LIN {X 0,Y 311.633,Z 530.648,A -85,B 0,C 180,E1 -15771.834,E2 -15771.834} C_VEL
LIN {X 0,Y 312.402,Z 526.953,A -85,B 0,C 180,E1 -15773.886,E2 -15773.886} C_VEL
LIN {X 0,Y 313.36,Z 522.43,A -85,B 0,C 180,E1 -15775.791,E2 -15775.791} C_VEL
LIN {X 0,Y 314.734,Z 515.773,A -85,B 0,C 180,E1 -15777.963,E2 -15777.963} C_VEL
LIN {X 0,Y 316.431,Z 507.874,A -85,B 0,C 180,E1 -15779.981,E2 -15779.981} C_VEL
LIN {X 0,Y 317.947,Z 499.641,A -85,B 0,C 180,E1 -15781.665,E2 -15781.665} C_VEL
LIN {X 0,Y 319.87,Z 489.513,A -85,B 0,C 180,E1 -15783.316,E2 -15783.316} C_VEL
LIN {X 0,Y 321.561,Z 479.498,A -85,B 0,C 180,E1 -15784.627,E2 -15784.627} C_VEL
LIN {X 0,Y 323.116,Z 468.579,A -85,B 0,C 180,E1 -15785.769,E2 -15785.769} C_VEL
LIN {X 0,Y 324.604,Z 456.019,A -85,B 0,C 180,E1 -15786.766,E2 -15786.766} C_VEL
LIN {X 0,Y 325.709,Z 443.241,A -85,B 0,C 180,E1 -15787.508,E2 -15787.508} C_VEL
LIN {X 0,Y 326.456,Z 430.389,A -85,B 0,C 180,E1 -15787.992,E2 -15787.992} C_VEL
LIN {X 0,Y 328.636,Z 357.959,A -85,B 0,C 180,E1 -15789.604,E2 -15789.604} C_VEL
LIN {X 0,Y 327.104,Z 351.684,A -85,B 0,C 180,E1 -15789.919,E2 -15789.919} C_VEL
LIN {X 0,Y 320.533,Z 336.835,A -85,B 0,C 180,E1 -15791,E2 -15791} C_VEL
LIN {X 0,Y 316.025,Z 327.77,A -85,B 0,C 180,E1 -15791.748,E2 -15791.748} C_VEL
LIN {X 0,Y 314.284,Z 325.682,A -85,B 0,C 180,E1 -15792.062,E2 -15792.062} C_VEL
LIN {X 0,Y 311.54,Z 323.906,A -85,B 0,C 180,E1 -15792.658,E2 -15792.658} C_VEL
LIN {X 0,Y 307.401,Z 321.61,A -85,B 0,C 180,E1 -15793.918,E2 -15793.918} C_VEL
LIN {X 0,Y 305.899,Z 319.461,A -85,B 0,C 180,E1 -15794.842,E2 -15794.842} C_VEL
LIN {X 0,Y 305.396,Z 317.446,A -85,B 0,C 180,E1 -15795.615,E2 -15795.615} C_VEL
LIN {X 0,Y 305.402,Z 317.444,A -85,B 0,C 180,E1 -15799.41,E2 -15799.41} C_VEL
LIN {X 0,Y 305.462,Z 317.438,A -85,B 0,C 180,E1 -15803.259,E2 -15803.259} C_VEL
LIN {X 0,Y 305.457,Z 317.413,A -85,B 0,C 180,E1 -15806.483,E2 -15806.483} C_VEL
LIN {X 0,Y 305.422,Z 317.44,A -85,B 0,C 180,E1 -15809.587,E2 -15809.587} C_VEL
LIN {X 0,Y 305.443,Z 317.437,A -85,B 0,C 180,E1 -15812.601,E2 -15812.601} C_VEL
LIN {X 0,Y 305.45,Z 317.436,A -85,B 0,C 180,E1 -15815.534,E2 -15815.534} C_VEL
LIN {X 0,Y 305.47,Z 317.436,A -85,B 0,C 180,E1 -15819.812,E2 -15819.812} C_VEL
LIN {X 0,Y 305.505,Z 317.43,A -85,B 0,C 180,E1 -15823.975,E2 -15823.975} C_VEL
LIN {X 0,Y 305.56,Z 317.41,A -85,B 0,C 180,E1 -15826.703,E2 -15826.703} C_VEL
LIN {X 0,Y 305.744,Z 317.386,A -85,B 0,C 180,E1 -15831.262,E2 -15831.262} C_VEL
LIN {X 0,Y 305.773,Z 317.392,A -85,B 0,C 180,E1 -15833.401,E2 -15833.401} C_VEL
LIN {X 0,Y 305.922,Z 317.377,A -85,B 0,C 180,E1 -15838.684,E2 -15838.684} C_VEL
LIN {X 0,Y 305.936,Z 317.367,A -85,B 0,C 180,E1 -15841.317,E2 -15841.317} C_VEL
LIN {X 0,Y 305.784,Z 317.385,A -85,B 0,C 180,E1 -15846.599,E2 -15846.599} C_VEL
LIN {X 0,Y 305.686,Z 317.401,A -85,B 0,C 180,E1 -15849.262,E2 -15849.262} C_VEL
LIN {X 0,Y 305.578,Z 317.405,A -85,B 0,C 180,E1 -15853.297,E2 -15853.297} C_VEL
LIN {X 0,Y 305.544,Z 317.42,A -85,B 0,C 180,E1 -15856.023,E2 -15856.023} C_VEL
LIN {X 0,Y 305.539,Z 317.417,A -85,B 0,C 180,E1 -15859.429,E2 -15859.429} C_VEL
LIN {X 0,Y 305.464,Z 317.423,A -85,B 0,C 180,E1 -15863.033,E2 -15863.033} C_VEL
LIN {X 0,Y 305.446,Z 317.433,A -85,B 0,C 180,E1 -15866.192,E2 -15866.192} C_VEL
LIN {X 0,Y 305.442,Z 317.435,A -85,B 0,C 180,E1 -15869.035,E2 -15869.035} C_VEL
LIN {X 0,Y 305.43,Z 317.432,A -85,B 0,C 180,E1 -15871.954,E2 -15871.954} C_VEL
LIN {X 0,Y 305.456,Z 317.431,A -85,B 0,C 180,E1 -15875.114,E2 -15875.114} C_VEL
LIN {X 0,Y 305.405,Z 317.437,A -85,B 0,C 180,E1 -15878.521,E2 -15878.521} C_VEL
LIN {X 0,Y 305.431,Z 317.422,A -85,B 0,C 180,E1 -15882.583,E2 -15882.583} C_VEL
LIN {X 0,Y 305.421,Z 317.445,A -85,B 0,C 180,E1 -15886.346,E2 -15886.346} C_VEL
LIN {X 0,Y 305.454,Z 317.439,A -85,B 0,C 180,E1 -15889.894,E2 -15889.894} C_VEL
LIN {X 0,Y 305.506,Z 317.511,A -85,B 0,C 180,E1 -15894.085,E2 -15894.085} C_VEL
LIN {X 0,Y 307.997,Z 327.276,A -85,B 0,C 180,E1 -15897.595,E2 -15897.595} C_VEL
LIN {X 0,Y 310.234,Z 336.989,A -85,B 0,C 180,E1 -15900.854,E2 -15900.854} C_VEL
LIN {X 0,Y 310.749,Z 339.325,A -85,B 0,C 180,E1 -15901.605,E2 -15901.605} C_VEL
LIN {X 0,Y 315.733,Z 351.12,A -85,B 0,C 180,E1 -15902.503,E2 -15902.503} C_VEL
LIN {X 0,Y 320.684,Z 375.641,A -85,B 0,C 180,E1 -15903.684,E2 -15903.684} C_VEL
LIN {X 0,Y 321.841,Z 383.222,A -85,B 0,C 180,E1 -15904,E2 -15904} C_VEL
LIN {X 0,Y 319.871,Z 448.323,A -85,B 0,C 180,E1 -15905.5,E2 -15905.5} C_VEL
LIN {X 0,Y 318.913,Z 461.298,A -85,B 0,C 180,E1 -15906.028,E2 -15906.028} C_VEL
LIN {X 0,Y 317.608,Z 472.761,A -85,B 0,C 180,E1 -15906.702,E2 -15906.702} C_VEL
LIN {X 0,Y 316.083,Z 484.24,A -85,B 0,C 180,E1 -15907.62,E2 -15907.62} C_VEL
LIN {X 0,Y 314.465,Z 494.745,A -85,B 0,C 180,E1 -15908.706,E2 -15908.706} C_VEL
LIN {X 0,Y 312.395,Z 505.538,A -85,B 0,C 180,E1 -15910.108,E2 -15910.108} C_VEL
LIN {X 0,Y 310.427,Z 515.474,A -85,B 0,C 180,E1 -15911.738,E2 -15911.738} C_VEL
LIN {X 0,Y 308.824,Z 523.96,A -85,B 0,C 180,E1 -15913.474,E2 -15913.474} C_VEL
LIN {X 0,Y 307.146,Z 531.649,A -85,B 0,C 180,E1 -15915.423,E2 -15915.423} C_VEL
LIN {X 0,Y 305.816,Z 537.841,A -85,B 0,C 180,E1 -15917.391,E2 -15917.391} C_VEL
LIN {X 0,Y 304.865,Z 542.782,A -85,B 0,C 180,E1 -15919.374,E2 -15919.374} C_VEL
LIN {X 0,Y 304.196,Z 546.618,A -85,B 0,C 180,E1 -15921.364,E2 -15921.364} C_VEL
LIN {X 0,Y 303.827,Z 549.45,A -85,B 0,C 180,E1 -15923.36,E2 -15923.36} C_VEL
LIN {X 0,Y 303.597,Z 551.759,A -85,B 0,C 180,E1 -15926.019,E2 -15926.019} C_VEL
LIN {X 0,Y 303.602,Z 552.335,A -85,B 0,C 180,E1 -15927.348,E2 -15927.348} C_VEL
LIN {X 0,Y 303.565,Z 552.482,A -85,B 0,C 180,E1 -15928.675,E2 -15928.675} C_VEL
LIN {X 0,Y 303.605,Z 552.23,A -85,B 0,C 180,E1 -15930.001,E2 -15930.001} C_VEL
LIN {X 0,Y 303.58,Z 551.589,A -85,B 0,C 180,E1 -15931.328,E2 -15931.328} C_VEL
LIN {X 0,Y 303.616,Z 550.557,A -85,B 0,C 180,E1 -15932.655,E2 -15932.655} C_VEL
LIN {X 0,Y 303.642,Z 549.076,A -85,B 0,C 180,E1 -15933.983,E2 -15933.983} C_VEL
LIN {X 0,Y 303.675,Z 546.624,A -85,B 0,C 180,E1 -15935.638,E2 -15935.638} C_VEL
LIN {X 0,Y 303.945,Z 541.933,A -85,B 0,C 180,E1 -15937.976,E2 -15937.976} C_VEL
LIN {X 0,Y 304.473,Z 535.613,A -85,B 0,C 180,E1 -15940.306,E2 -15940.306} C_VEL
LIN {X 0,Y 305.198,Z 528.715,A -85,B 0,C 180,E1 -15942.3,E2 -15942.3} C_VEL
LIN {X 0,Y 306.095,Z 521.67,A -85,B 0,C 180,E1 -15943.952,E2 -15943.952} C_VEL
LIN {X 0,Y 307.18,Z 513.169,A -85,B 0,C 180,E1 -15945.596,E2 -15945.596} C_VEL
LIN {X 0,Y 308.266,Z 502.616,A -85,B 0,C 180,E1 -15947.241,E2 -15947.241} C_VEL
LIN {X 0,Y 309.485,Z 492.181,A -85,B 0,C 180,E1 -15948.538,E2 -15948.538} C_VEL
LIN {X 0,Y 310.709,Z 480.737,A -85,B 0,C 180,E1 -15949.662,E2 -15949.662} C_VEL
LIN {X 0,Y 311.763,Z 468.97,A -85,B 0,C 180,E1 -15950.539,E2 -15950.539} C_VEL
LIN {X 0,Y 312.642,Z 455.38,A -85,B 0,C 180,E1 -15951.254,E2 -15951.254} C_VEL
LIN {X 0,Y 313.173,Z 441.759,A -85,B 0,C 180,E1 -15951.691,E2 -15951.691} C_VEL
LIN {X 0,Y 314.389,Z 380.153,A -85,B 0,C 180,E1 -15953.088,E2 -15953.088} C_VEL
LIN {X 0,Y 308.852,Z 339.998,A -85,B 0,C 180,E1 -15954.446,E2 -15954.446} C_VEL
LIN {X 0,Y 309.01,Z 335.76,A -85,B 0,C 180,E1 -15955.604,E2 -15955.604} C_VEL
LIN {X 0,Y 307.372,Z 326.429,A -85,B 0,C 180,E1 -15958.324,E2 -15958.324} C_VEL
LIN {X 0,Y 305.509,Z 317.433,A -85,B 0,C 180,E1 -15961.076,E2 -15961.076} C_VEL
LIN {X 0,Y 305.466,Z 317.433,A -85,B 0,C 180,E1 -15965.114,E2 -15965.114} C_VEL
LIN {X 0,Y 305.416,Z 317.441,A -85,B 0,C 180,E1 -15968.52,E2 -15968.52} C_VEL
LIN {X 0,Y 305.44,Z 317.439,A -85,B 0,C 180,E1 -15972.582,E2 -15972.582} C_VEL
LIN {X 0,Y 305.43,Z 317.442,A -85,B 0,C 180,E1 -15976.345,E2 -15976.345} C_VEL
LIN {X 0,Y 305.463,Z 317.433,A -85,B 0,C 180,E1 -15979.893,E2 -15979.893} C_VEL
LIN {X 0,Y 305.485,Z 317.429,A -85,B 0,C 180,E1 -15983.632,E2 -15983.632} C_VEL
LIN {X 0,Y 305.47,Z 317.433,A -85,B 0,C 180,E1 -15986.483,E2 -15986.483} C_VEL
LIN {X 0,Y 305.439,Z 317.435,A -85,B 0,C 180,E1 -15989.588,E2 -15989.588} C_VEL
LIN {X 0,Y 305.476,Z 317.432,A -85,B 0,C 180,E1 -15992.604,E2 -15992.604} C_VEL
LIN {X 0,Y 305.493,Z 317.43,A -85,B 0,C 180,E1 -15995.537,E2 -15995.537} C_VEL
LIN {X 0,Y 305.489,Z 317.425,A -85,B 0,C 180,E1 -15999.813,E2 -15999.813} C_VEL
LIN {X 0,Y 305.555,Z 317.422,A -85,B 0,C 180,E1 -16003.978,E2 -16003.978} C_VEL
LIN {X 0,Y 305.591,Z 317.415,A -85,B 0,C 180,E1 -16006.704,E2 -16006.704} C_VEL
LIN {X 0,Y 305.76,Z 317.389,A -85,B 0,C 180,E1 -16011.258,E2 -16011.258} C_VEL
LIN {X 0,Y 305.811,Z 317.387,A -85,B 0,C 180,E1 -16013.401,E2 -16013.401} C_VEL
LIN {X 0,Y 305.953,Z 317.37,A -85,B 0,C 180,E1 -16018.683,E2 -16018.683} C_VEL
LIN {X 0,Y 305.954,Z 317.365,A -85,B 0,C 180,E1 -16021.316,E2 -16021.316} C_VEL
LIN {X 0,Y 305.67,Z 317.403,A -85,B 0,C 180,E1 -16025.277,E2 -16025.277} C_VEL
LIN {X 0,Y 305.75,Z 317.397,A -85,B 0,C 180,E1 -16027.927,E2 -16027.927} C_VEL
LIN {X 0,Y 305.603,Z 317.413,A -85,B 0,C 180,E1 -16031.945,E2 -16031.945} C_VEL
LIN {X 0,Y 305.612,Z 317.408,A -85,B 0,C 180,E1 -16035.014,E2 -16035.014} C_VEL
LIN {X 0,Y 305.521,Z 317.427,A -85,B 0,C 180,E1 -16038.786,E2 -16038.786} C_VEL
LIN {X 0,Y 305.49,Z 317.432,A -85,B 0,C 180,E1 -16043.039,E2 -16043.039} C_VEL
LIN {X 0,Y 305.481,Z 317.425,A -85,B 0,C 180,E1 -16046.2,E2 -16046.2} C_VEL
LIN {X 0,Y 305.466,Z 317.428,A -85,B 0,C 180,E1 -16049.038,E2 -16049.038} C_VEL
LIN {X 0,Y 305.44,Z 317.434,A -85,B 0,C 180,E1 -16051.952,E2 -16051.952} C_VEL
LIN {X 0,Y 305.465,Z 317.433,A -85,B 0,C 180,E1 -16055.112,E2 -16055.112} C_VEL
LIN {X 0,Y 305.443,Z 317.427,A -85,B 0,C 180,E1 -16058.526,E2 -16058.526} C_VEL
LIN {X 0,Y 305.457,Z 317.432,A -85,B 0,C 180,E1 -16062.585,E2 -16062.585} C_VEL
LIN {X 0,Y 305.427,Z 317.434,A -85,B 0,C 180,E1 -16066.344,E2 -16066.344} C_VEL
LIN {X 0,Y 305.459,Z 317.435,A -85,B 0,C 180,E1 -16069.891,E2 -16069.891} C_VEL
LIN {X 0,Y 305.465,Z 317.432,A -85,B 0,C 180,E1 -16073.635,E2 -16073.635} C_VEL
LIN {X 0,Y 305.467,Z 317.435,A -85,B 0,C 180,E1 -16076.482,E2 -16076.482} C_VEL
LIN {X 0,Y 305.444,Z 317.434,A -85,B 0,C 180,E1 -16079.588,E2 -16079.588} C_VEL
LIN {X 0,Y 305.473,Z 317.436,A -85,B 0,C 180,E1 -16082.603,E2 -16082.603} C_VEL
LIN {X 0,Y 305.493,Z 317.428,A -85,B 0,C 180,E1 -16085.536,E2 -16085.536} C_VEL
LIN {X 0,Y 305.514,Z 317.427,A -85,B 0,C 180,E1 -16089.814,E2 -16089.814} C_VEL
LIN {X 0,Y 305.545,Z 317.426,A -85,B 0,C 180,E1 -16092.6,E2 -16092.6} C_VEL
LIN {X 0,Y 305.627,Z 317.415,A -85,B 0,C 180,E1 -16095.347,E2 -16095.347} C_VEL
LIN {X 0,Y 305.649,Z 317.603,A -85,B 0,C 180,E1 -16097.381,E2 -16097.381} C_VEL
LIN {X 0,Y 307.014,Z 324.322,A -85,B 0,C 180,E1 -16099.514,E2 -16099.514} C_VEL
LIN {X 0,Y 311.663,Z 338.303,A -85,B 0,C 180,E1 -16100.189,E2 -16100.189} C_VEL
LIN {X 0,Y 314.867,Z 355.721,A -85,B 0,C 180,E1 -16100.816,E2 -16100.816} C_VEL
LIN {X 0,Y 313.102,Z 432.447,A -85,B 0,C 180,E1 -16102.583,E2 -16102.583} C_VEL
LIN {X 0,Y 312.504,Z 444.643,A -85,B 0,C 180,E1 -16103.097,E2 -16103.097} C_VEL
LIN {X 0,Y 311.661,Z 457.936,A -85,B 0,C 180,E1 -16103.931,E2 -16103.931} C_VEL
LIN {X 0,Y 310.641,Z 469.932,A -85,B 0,C 180,E1 -16104.971,E2 -16104.971} C_VEL
LIN {X 0,Y 309.465,Z 481.372,A -85,B 0,C 180,E1 -16106.255,E2 -16106.255} C_VEL
LIN {X 0,Y 308.21,Z 491.721,A -85,B 0,C 180,E1 -16107.712,E2 -16107.712} C_VEL
LIN {X 0,Y 307.015,Z 501.006,A -85,B 0,C 180,E1 -16109.343,E2 -16109.343} C_VEL
LIN {X 0,Y 305.866,Z 510.01,A -85,B 0,C 180,E1 -16111.315,E2 -16111.315} C_VEL
LIN {X 0,Y 305.023,Z 517.26,A -85,B 0,C 180,E1 -16113.301,E2 -16113.301} C_VEL
LIN {X 0,Y 304.453,Z 523.042,A -85,B 0,C 180,E1 -16115.297,E2 -16115.297} C_VEL
LIN {X 0,Y 304.041,Z 527.598,A -85,B 0,C 180,E1 -16117.303,E2 -16117.303} C_VEL
LIN {X 0,Y 303.699,Z 531.071,A -85,B 0,C 180,E1 -16119.321,E2 -16119.321} C_VEL
LIN {X 0,Y 303.515,Z 532.798,A -85,B 0,C 180,E1 -16120.674,E2 -16120.674} C_VEL
LIN {X 0,Y 303.468,Z 534.112,A -85,B 0,C 180,E1 -16122.029,E2 -16122.029} C_VEL
LIN {X 0,Y 303.461,Z 535.04,A -85,B 0,C 180,E1 -16123.421,E2 -16123.421} C_VEL
LIN {X 0,Y 303.436,Z 535.485,A -85,B 0,C 180,E1 -16124.759,E2 -16124.759} C_VEL
LIN {X 0,Y 303.462,Z 535.535,A -85,B 0,C 180,E1 -16126.134,E2 -16126.134} C_VEL
LIN {X 0,Y 303.807,Z 534.666,A -85,B 0,C 180,E1 -16128.477,E2 -16128.477} C_VEL
LIN {X 0,Y 304.097,Z 533.152,A -85,B 0,C 180,E1 -16130.282,E2 -16130.282} C_VEL
LIN {X 0,Y 304.9,Z 529.796,A -85,B 0,C 180,E1 -16132.78,E2 -16132.78} C_VEL
LIN {X 0,Y 305.907,Z 525.122,A -85,B 0,C 180,E1 -16135.151,E2 -16135.151} C_VEL
LIN {X 0,Y 307.165,Z 519.622,A -85,B 0,C 180,E1 -16137.231,E2 -16137.231} C_VEL
LIN {X 0,Y 308.709,Z 512.642,A -85,B 0,C 180,E1 -16139.304,E2 -16139.304} C_VEL
LIN {X 0,Y 310.269,Z 505.274,A -85,B 0,C 180,E1 -16141.06,E2 -16141.06} C_VEL
LIN {X 0,Y 312.033,Z 496.703,A -85,B 0,C 180,E1 -16142.72,E2 -16142.72} C_VEL
LIN {X 0,Y 313.87,Z 486.979,A -85,B 0,C 180,E1 -16144.233,E2 -16144.233} C_VEL
LIN {X 0,Y 315.659,Z 476.269,A -85,B 0,C 180,E1 -16145.566,E2 -16145.566} C_VEL
LIN {X 0,Y 317.333,Z 464.433,A -85,B 0,C 180,E1 -16146.723,E2 -16146.723} C_VEL
LIN {X 0,Y 318.661,Z 453.162,A -85,B 0,C 180,E1 -16147.555,E2 -16147.555} C_VEL
LIN {X 0,Y 319.643,Z 440.318,A -85,B 0,C 180,E1 -16148.247,E2 -16148.247} C_VEL
LIN {X 0,Y 320.384,Z 426.831,A -85,B 0,C 180,E1 -16148.694,E2 -16148.694} C_VEL
LIN {X 0,Y 322.483,Z 359.121,A -85,B 0,C 180,E1 -16150.213,E2 -16150.213} C_VEL
LIN {X 0,Y 321.121,Z 354.046,A -85,B 0,C 180,E1 -16150.489,E2 -16150.489} C_VEL
LIN {X 0,Y 314.427,Z 338.884,A -85,B 0,C 180,E1 -16151.636,E2 -16151.636} C_VEL
LIN {X 0,Y 307.332,Z 324.798,A -85,B 0,C 180,E1 -16152.885,E2 -16152.885} C_VEL
LIN {X 0,Y 305.899,Z 319.461,A -85,B 0,C 180,E1 -16154.842,E2 -16154.842} C_VEL
LIN {X 0,Y 305.177,Z 318.215,A -85,B 0,C 180,E1 -16155.513,E2 -16155.513} C_VEL
LIN {X 0,Y 304.125,Z 317.72,A -85,B 0,C 180,E1 -16156.21,E2 -16156.21} C_VEL
LIN {X 0,Y 299.351,Z 318.22,A -85,B 0,C 180,E1 -16159.117,E2 -16159.117} C_VEL
LIN {X 0,Y 298.434,Z 318.312,A -85,B 0,C 180,E1 -16160.266,E2 -16160.266} C_VEL
LIN {X 0,Y 298.367,Z 318.32,A -85,B 0,C 180,E1 -16160.653,E2 -16160.653} C_VEL
LIN {X 0,Y 298.409,Z 318.315,A -85,B 0,C 180,E1 -16163.929,E2 -16163.929} C_VEL
LIN {X 0,Y 298.385,Z 318.298,A -85,B 0,C 180,E1 -16167.199,E2 -16167.199} C_VEL
LIN {X 0,Y 298.394,Z 318.309,A -85,B 0,C 180,E1 -16170.625,E2 -16170.625} C_VEL
LIN {X 0,Y 298.415,Z 318.308,A -85,B 0,C 180,E1 -16174.918,E2 -16174.918} C_VEL
LIN {X 0,Y 298.389,Z 318.308,A -85,B 0,C 180,E1 -16177.862,E2 -16177.862} C_VEL
LIN {X 0,Y 298.451,Z 318.306,A -85,B 0,C 180,E1 -16180.751,E2 -16180.751} C_VEL
LIN {X 0,Y 298.502,Z 318.299,A -85,B 0,C 180,E1 -16184.99,E2 -16184.99} C_VEL
LIN {X 0,Y 298.572,Z 318.291,A -85,B 0,C 180,E1 -16189.146,E2 -16189.146} C_VEL
LIN {X 0,Y 298.687,Z 318.265,A -85,B 0,C 180,E1 -16191.884,E2 -16191.884} C_VEL
LIN {X 0,Y 298.614,Z 318.286,A -85,B 0,C 180,E1 -16194.598,E2 -16194.598} C_VEL
LIN {X 0,Y 298.889,Z 318.252,A -85,B 0,C 180,E1 -16198.653,E2 -16198.653} C_VEL
LIN {X 0,Y 298.902,Z 318.243,A -85,B 0,C 180,E1 -16201.348,E2 -16201.348} C_VEL
LIN {X 0,Y 298.732,Z 318.262,A -85,B 0,C 180,E1 -16206.756,E2 -16206.756} C_VEL
LIN {X 0,Y 298.617,Z 318.283,A -85,B 0,C 180,E1 -16209.483,E2 -16209.483} C_VEL
LIN {X 0,Y 298.537,Z 318.282,A -85,B 0,C 180,E1 -16213.616,E2 -16213.616} C_VEL
LIN {X 0,Y 298.48,Z 318.302,A -85,B 0,C 180,E1 -16216.413,E2 -16216.413} C_VEL
LIN {X 0,Y 298.479,Z 318.299,A -85,B 0,C 180,E1 -16219.642,E2 -16219.642} C_VEL
LIN {X 0,Y 298.403,Z 318.304,A -85,B 0,C 180,E1 -16223.603,E2 -16223.603} C_VEL
LIN {X 0,Y 298.396,Z 318.311,A -85,B 0,C 180,E1 -16226.584,E2 -16226.584} C_VEL
LIN {X 0,Y 298.387,Z 318.318,A -85,B 0,C 180,E1 -16229.645,E2 -16229.645} C_VEL
LIN {X 0,Y 298.387,Z 318.313,A -85,B 0,C 180,E1 -16232.802,E2 -16232.802} C_VEL
LIN {X 0,Y 298.421,Z 318.311,A -85,B 0,C 180,E1 -16236.804,E2 -16236.804} C_VEL
LIN {X 0,Y 298.343,Z 318.321,A -85,B 0,C 180,E1 -16241.269,E2 -16241.269} C_VEL
LIN {X 0,Y 298.35,Z 318.314,A -85,B 0,C 180,E1 -16245.036,E2 -16245.036} C_VEL
LIN {X 0,Y 298.381,Z 318.323,A -85,B 0,C 180,E1 -16248.74,E2 -16248.74} C_VEL
LIN {X 0,Y 298.405,Z 318.317,A -85,B 0,C 180,E1 -16252.242,E2 -16252.242} C_VEL
LIN {X 0,Y 298.447,Z 318.348,A -85,B 0,C 180,E1 -16253.284,E2 -16253.284} C_VEL
LIN {X 0,Y 300.783,Z 327.365,A -85,B 0,C 180,E1 -16256.656,E2 -16256.656} C_VEL
LIN {X 0,Y 303.273,Z 337.968,A -85,B 0,C 180,E1 -16260.344,E2 -16260.344} C_VEL
LIN {X 0,Y 303.564,Z 339.259,A -85,B 0,C 180,E1 -16260.719,E2 -16260.719} C_VEL
LIN {X 0,Y 309.944,Z 353.535,A -85,B 0,C 180,E1 -16261.898,E2 -16261.898} C_VEL
LIN {X 0,Y 314.772,Z 378.069,A -85,B 0,C 180,E1 -16263.109,E2 -16263.109} C_VEL
LIN {X 0,Y 315.699,Z 384.414,A -85,B 0,C 180,E1 -16263.378,E2 -16263.378} C_VEL
LIN {X 0,Y 313.715,Z 447.58,A -85,B 0,C 180,E1 -16264.854,E2 -16264.854} C_VEL
LIN {X 0,Y 312.74,Z 460.729,A -85,B 0,C 180,E1 -16265.391,E2 -16265.391} C_VEL
LIN {X 0,Y 311.294,Z 472.851,A -85,B 0,C 180,E1 -16266.112,E2 -16266.112} C_VEL
LIN {X 0,Y 309.581,Z 485.097,A -85,B 0,C 180,E1 -16267.124,E2 -16267.124} C_VEL
LIN {X 0,Y 307.609,Z 496.652,A -85,B 0,C 180,E1 -16268.384,E2 -16268.384} C_VEL
LIN {X 0,Y 305.545,Z 507.071,A -85,B 0,C 180,E1 -16269.818,E2 -16269.818} C_VEL
LIN {X 0,Y 303.399,Z 517.146,A -85,B 0,C 180,E1 -16271.57,E2 -16271.57} C_VEL
LIN {X 0,Y 301.736,Z 525.561,A -85,B 0,C 180,E1 -16273.423,E2 -16273.423} C_VEL
LIN {X 0,Y 300.038,Z 532.905,A -85,B 0,C 180,E1 -16275.417,E2 -16275.417} C_VEL
LIN {X 0,Y 298.499,Z 539.692,A -85,B 0,C 180,E1 -16277.768,E2 -16277.768} C_VEL
LIN {X 0,Y 297.589,Z 544.192,A -85,B 0,C 180,E1 -16279.799,E2 -16279.799} C_VEL
LIN {X 0,Y 296.98,Z 547.633,A -85,B 0,C 180,E1 -16281.838,E2 -16281.838} C_VEL
LIN {X 0,Y 296.553,Z 550.614,A -85,B 0,C 180,E1 -16284.481,E2 -16284.481} C_VEL
LIN {X 0,Y 296.499,Z 551.619,A -85,B 0,C 180,E1 -16285.924,E2 -16285.924} C_VEL
LIN {X 0,Y 296.527,Z 552.16,A -85,B 0,C 180,E1 -16287.284,E2 -16287.284} C_VEL
LIN {X 0,Y 296.52,Z 551.995,A -85,B 0,C 180,E1 -16290.001,E2 -16290.001} C_VEL
LIN {X 0,Y 296.499,Z 551.331,A -85,B 0,C 180,E1 -16291.359,E2 -16291.359} C_VEL
LIN {X 0,Y 296.542,Z 550.268,A -85,B 0,C 180,E1 -16292.718,E2 -16292.718} C_VEL
LIN {X 0,Y 296.541,Z 548.743,A -85,B 0,C 180,E1 -16294.078,E2 -16294.078} C_VEL
LIN {X 0,Y 296.622,Z 545.657,A -85,B 0,C 180,E1 -16296.121,E2 -16296.121} C_VEL
LIN {X 0,Y 296.88,Z 541.491,A -85,B 0,C 180,E1 -16298.167,E2 -16298.167} C_VEL
LIN {X 0,Y 297.445,Z 535.109,A -85,B 0,C 180,E1 -16300.552,E2 -16300.552} C_VEL
LIN {X 0,Y 298.225,Z 528.144,A -85,B 0,C 180,E1 -16302.592,E2 -16302.592} C_VEL
LIN {X 0,Y 299.129,Z 521.018,A -85,B 0,C 180,E1 -16304.283,E2 -16304.283} C_VEL
LIN {X 0,Y 300.285,Z 512.398,A -85,B 0,C 180,E1 -16305.963,E2 -16305.963} C_VEL
LIN {X 0,Y 301.423,Z 501.704,A -85,B 0,C 180,E1 -16307.646,E2 -16307.646} C_VEL
LIN {X 0,Y 302.685,Z 491.116,A -85,B 0,C 180,E1 -16308.971,E2 -16308.971} C_VEL
LIN {X 0,Y 303.978,Z 479.4,A -85,B 0,C 180,E1 -16310.116,E2 -16310.116} C_VEL
LIN {X 0,Y 305.071,Z 467.2,A -85,B 0,C 180,E1 -16311.01,E2 -16311.01} C_VEL
LIN {X 0,Y 305.957,Z 453.904,A -85,B 0,C 180,E1 -16311.697,E2 -16311.697} C_VEL
LIN {X 0,Y 306.425,Z 440.846,A -85,B 0,C 180,E1 -16312.105,E2 -16312.105} C_VEL
LIN {X 0,Y 307.664,Z 380.712,A -85,B 0,C 180,E1 -16313.497,E2 -16313.497} C_VEL
LIN {X 0,Y 301.977,Z 339.873,A -85,B 0,C 180,E1 -16314.899,E2 -16314.899} C_VEL
LIN {X 0,Y 302.008,Z 336.556,A -85,B 0,C 180,E1 -16315.834,E2 -16315.834} C_VEL
LIN {X 0,Y 300.285,Z 327.076,A -85,B 0,C 180,E1 -16318.673,E2 -16318.673} C_VEL
LIN {X 0,Y 298.425,Z 318.31,A -85,B 0,C 180,E1 -16321.422,E2 -16321.422} C_VEL
LIN {X 0,Y 298.433,Z 318.31,A -85,B 0,C 180,E1 -16324.488,E2 -16324.488} C_VEL
LIN {X 0,Y 298.391,Z 318.317,A -85,B 0,C 180,E1 -16327.763,E2 -16327.763} C_VEL
LIN {X 0,Y 298.352,Z 318.319,A -85,B 0,C 180,E1 -16331.268,E2 -16331.268} C_VEL
LIN {X 0,Y 298.359,Z 318.319,A -85,B 0,C 180,E1 -16335.035,E2 -16335.035} C_VEL
LIN {X 0,Y 298.389,Z 318.318,A -85,B 0,C 180,E1 -16338.739,E2 -16338.739} C_VEL
LIN {X 0,Y 298.412,Z 318.312,A -85,B 0,C 180,E1 -16342.241,E2 -16342.241} C_VEL
LIN {X 0,Y 298.413,Z 318.31,A -85,B 0,C 180,E1 -16345.581,E2 -16345.581} C_VEL
LIN {X 0,Y 298.384,Z 318.318,A -85,B 0,C 180,E1 -16348.79,E2 -16348.79} C_VEL
LIN {X 0,Y 298.431,Z 318.308,A -85,B 0,C 180,E1 -16351.901,E2 -16351.901} C_VEL
LIN {X 0,Y 298.455,Z 318.308,A -85,B 0,C 180,E1 -16354.921,E2 -16354.921} C_VEL
LIN {X 0,Y 298.419,Z 318.308,A -85,B 0,C 180,E1 -16357.863,E2 -16357.863} C_VEL
LIN {X 0,Y 298.482,Z 318.296,A -85,B 0,C 180,E1 -16360.753,E2 -16360.753} C_VEL
LIN {X 0,Y 298.591,Z 318.289,A -85,B 0,C 180,E1 -16364.994,E2 -16364.994} C_VEL
LIN {X 0,Y 298.596,Z 318.285,A -85,B 0,C 180,E1 -16369.146,E2 -16369.146} C_VEL
LIN {X 0,Y 298.722,Z 318.27,A -85,B 0,C 180,E1 -16371.885,E2 -16371.885} C_VEL
LIN {X 0,Y 298.645,Z 318.281,A -85,B 0,C 180,E1 -16374.598,E2 -16374.598} C_VEL
LIN {X 0,Y 298.92,Z 318.246,A -85,B 0,C 180,E1 -16378.652,E2 -16378.652} C_VEL
LIN {X 0,Y 298.921,Z 318.241,A -85,B 0,C 180,E1 -16381.347,E2 -16381.347} C_VEL
LIN {X 0,Y 298.713,Z 318.272,A -85,B 0,C 180,E1 -16386.542,E2 -16386.542} C_VEL
LIN {X 0,Y 298.629,Z 318.283,A -85,B 0,C 180,E1 -16389.482,E2 -16389.482} C_VEL
LIN {X 0,Y 298.549,Z 318.287,A -85,B 0,C 180,E1 -16393.615,E2 -16393.615} C_VEL
LIN {X 0,Y 298.488,Z 318.295,A -85,B 0,C 180,E1 -16396.412,E2 -16396.412} C_VEL
LIN {X 0,Y 298.463,Z 318.303,A -85,B 0,C 180,E1 -16399.626,E2 -16399.626} C_VEL
LIN {X 0,Y 298.428,Z 318.307,A -85,B 0,C 180,E1 -16403.6,E2 -16403.6} C_VEL
LIN {X 0,Y 298.42,Z 318.305,A -85,B 0,C 180,E1 -16406.581,E2 -16406.581} C_VEL
LIN {X 0,Y 298.403,Z 318.31,A -85,B 0,C 180,E1 -16409.643,E2 -16409.643} C_VEL
LIN {X 0,Y 298.396,Z 318.312,A -85,B 0,C 180,E1 -16412.8,E2 -16412.8} C_VEL
LIN {X 0,Y 298.447,Z 318.302,A -85,B 0,C 180,E1 -16416.806,E2 -16416.806} C_VEL
LIN {X 0,Y 298.389,Z 318.311,A -85,B 0,C 180,E1 -16421.087,E2 -16421.087} C_VEL
LIN {X 0,Y 298.401,Z 318.312,A -85,B 0,C 180,E1 -16423.102,E2 -16423.102} C_VEL
LIN {X 0,Y 298.405,Z 318.306,A -85,B 0,C 180,E1 -16426.92,E2 -16426.92} C_VEL
LIN {X 0,Y 298.392,Z 318.313,A -85,B 0,C 180,E1 -16431.009,E2 -16431.009} C_VEL
LIN {X 0,Y 298.407,Z 318.313,A -85,B 0,C 180,E1 -16433.927,E2 -16433.927} C_VEL
LIN {X 0,Y 298.395,Z 318.312,A -85,B 0,C 180,E1 -16437.199,E2 -16437.199} C_VEL
LIN {X 0,Y 298.416,Z 318.314,A -85,B 0,C 180,E1 -16440.62,E2 -16440.62} C_VEL
LIN {X 0,Y 298.453,Z 318.308,A -85,B 0,C 180,E1 -16444.92,E2 -16444.92} C_VEL
LIN {X 0,Y 298.448,Z 318.308,A -85,B 0,C 180,E1 -16449.314,E2 -16449.314} C_VEL
LIN {X 0,Y 298.51,Z 318.3,A -85,B 0,C 180,E1 -16452.177,E2 -16452.177} C_VEL
LIN {X 0,Y 298.586,Z 318.293,A -85,B 0,C 180,E1 -16454.993,E2 -16454.993} C_VEL
LIN {X 0,Y 298.549,Z 318.305,A -85,B 0,C 180,E1 -16456.99,E2 -16456.99} C_VEL
LIN {X 0,Y 299.873,Z 324.691,A -85,B 0,C 180,E1 -16459.039,E2 -16459.039} C_VEL
LIN {X 0,Y 305.319,Z 340.966,A -85,B 0,C 180,E1 -16459.829,E2 -16459.829} C_VEL
LIN {X 0,Y 308.171,Z 356.686,A -85,B 0,C 180,E1 -16460.407,E2 -16460.407} C_VEL
LIN {X 0,Y 306.353,Z 432.063,A -85,B 0,C 180,E1 -16462.17,E2 -16462.17} C_VEL
LIN {X 0,Y 305.681,Z 445.217,A -85,B 0,C 180,E1 -16462.734,E2 -16462.734} C_VEL
LIN {X 0,Y 304.864,Z 457.85,A -85,B 0,C 180,E1 -16463.546,E2 -16463.546} C_VEL
LIN {X 0,Y 303.843,Z 469.705,A -85,B 0,C 180,E1 -16464.585,E2 -16464.585} C_VEL
LIN {X 0,Y 302.68,Z 480.632,A -85,B 0,C 180,E1 -16465.821,E2 -16465.821} C_VEL
LIN {X 0,Y 301.388,Z 491.243,A -85,B 0,C 180,E1 -16467.326,E2 -16467.326} C_VEL
LIN {X 0,Y 300.136,Z 500.687,A -85,B 0,C 180,E1 -16468.993,E2 -16468.993} C_VEL
LIN {X 0,Y 298.908,Z 509.783,A -85,B 0,C 180,E1 -16471.009,E2 -16471.009} C_VEL
LIN {X 0,Y 298.023,Z 517.106,A -85,B 0,C 180,E1 -16473.04,E2 -16473.04} C_VEL
LIN {X 0,Y 297.435,Z 522.067,A -85,B 0,C 180,E1 -16474.743,E2 -16474.743} C_VEL
LIN {X 0,Y 297.059,Z 526.875,A -85,B 0,C 180,E1 -16476.792,E2 -16476.792} C_VEL
LIN {X 0,Y 296.678,Z 530.579,A -85,B 0,C 180,E1 -16478.856,E2 -16478.856} C_VEL
LIN {X 0,Y 296.408,Z 533.253,A -85,B 0,C 180,E1 -16480.933,E2 -16480.933} C_VEL
LIN {X 0,Y 296.356,Z 535.245,A -85,B 0,C 180,E1 -16483.517,E2 -16483.517} C_VEL
LIN {X 0,Y 296.344,Z 535.717,A -85,B 0,C 180,E1 -16485.12,E2 -16485.12} C_VEL
LIN {X 0,Y 296.394,Z 535.71,A -85,B 0,C 180,E1 -16486.53,E2 -16486.53} C_VEL
LIN {X 0,Y 296.751,Z 534.87,A -85,B 0,C 180,E1 -16488.68,E2 -16488.68} C_VEL
LIN {X 0,Y 297.141,Z 533.095,A -85,B 0,C 180,E1 -16490.779,E2 -16490.779} C_VEL
LIN {X 0,Y 297.923,Z 530.023,A -85,B 0,C 180,E1 -16493.073,E2 -16493.073} C_VEL
LIN {X 0,Y 298.755,Z 526.335,A -85,B 0,C 180,E1 -16495.05,E2 -16495.05} C_VEL
LIN {X 0,Y 300.169,Z 520.546,A -85,B 0,C 180,E1 -16497.401,E2 -16497.401} C_VEL
LIN {X 0,Y 301.885,Z 513.258,A -85,B 0,C 180,E1 -16499.649,E2 -16499.649} C_VEL
LIN {X 0,Y 303.48,Z 506.133,A -85,B 0,C 180,E1 -16501.407,E2 -16501.407} C_VEL
LIN {X 0,Y 304.92,Z 499.369,A -85,B 0,C 180,E1 -16502.794,E2 -16502.794} C_VEL
LIN {X 0,Y 307.044,Z 489.078,A -85,B 0,C 180,E1 -16504.512,E2 -16504.512} C_VEL
LIN {X 0,Y 308.882,Z 478.928,A -85,B 0,C 180,E1 -16505.864,E2 -16505.864} C_VEL
LIN {X 0,Y 310.59,Z 467.688,A -85,B 0,C 180,E1 -16507.045,E2 -16507.045} C_VEL
LIN {X 0,Y 312.227,Z 454.894,A -85,B 0,C 180,E1 -16508.063,E2 -16508.063} C_VEL
LIN {X 0,Y 313.331,Z 442.514,A -85,B 0,C 180,E1 -16508.778,E2 -16508.778} C_VEL
LIN {X 0,Y 314.076,Z 430.21,A -85,B 0,C 180,E1 -16509.238,E2 -16509.238} C_VEL
LIN {X 0,Y 316.361,Z 360.241,A -85,B 0,C 180,E1 -16510.848,E2 -16510.848} C_VEL
LIN {X 0,Y 315.067,Z 356.085,A -85,B 0,C 180,E1 -16511.103,E2 -16511.103} C_VEL
LIN {X 0,Y 308.682,Z 341.783,A -85,B 0,C 180,E1 -16512.238,E2 -16512.238} C_VEL
LIN {X 0,Y 301.592,Z 328.083,A -85,B 0,C 180,E1 -16513.515,E2 -16513.515} C_VEL
LIN {X 0,Y 300.125,Z 325.054,A -85,B 0,C 180,E1 -16513.801,E2 -16513.801} C_VEL
LIN {X 0,Y 298.377,Z 318.311,A -85,B 0,C 180,E1 -16516.454,E2 -16516.454} C_VEL
LIN {X 0,Y 298.367,Z 318.32,A -85,B 0,C 180,E1 -16520.653,E2 -16520.653} C_VEL
LIN {X 0,Y 297.72,Z 318.406,A -85,B 0,C 180,E1 -16521.781,E2 -16521.781} C_VEL
LIN {X 0,Y 294.886,Z 318.756,A -85,B 0,C 180,E1 -16523.617,E2 -16523.617} C_VEL
LIN {X 0,Y 292.464,Z 319.039,A -85,B 0,C 180,E1 -16525.106,E2 -16525.106} C_VEL
LIN {X 0,Y 291.412,Z 319.161,A -85,B 0,C 180,E1 -16526.26,E2 -16526.26} C_VEL
LIN {X 0,Y 291.32,Z 319.173,A -85,B 0,C 180,E1 -16526.651,E2 -16526.651} C_VEL
LIN {X 0,Y 291.357,Z 319.186,A -85,B 0,C 180,E1 -16530.267,E2 -16530.267} C_VEL
LIN {X 0,Y 291.339,Z 319.187,A -85,B 0,C 180,E1 -16534.265,E2 -16534.265} C_VEL
LIN {X 0,Y 291.349,Z 319.187,A -85,B 0,C 180,E1 -16537.297,E2 -16537.297} C_VEL
LIN {X 0,Y 291.381,Z 319.188,A -85,B 0,C 180,E1 -16540.265,E2 -16540.265} C_VEL
LIN {X 0,Y 291.465,Z 319.176,A -85,B 0,C 180,E1 -16544.682,E2 -16544.682} C_VEL
LIN {X 0,Y 291.517,Z 319.17,A -85,B 0,C 180,E1 -16548.88,E2 -16548.88} C_VEL
LIN {X 0,Y 291.641,Z 319.141,A -85,B 0,C 180,E1 -16551.687,E2 -16551.687} C_VEL
LIN {X 0,Y 291.585,Z 319.162,A -85,B 0,C 180,E1 -16554.468,E2 -16554.468} C_VEL
LIN {X 0,Y 291.857,Z 319.127,A -85,B 0,C 180,E1 -16558.62,E2 -16558.62} C_VEL
LIN {X 0,Y 291.868,Z 319.118,A -85,B 0,C 180,E1 -16561.38,E2 -16561.38} C_VEL
LIN {X 0,Y 291.683,Z 319.138,A -85,B 0,C 180,E1 -16566.92,E2 -16566.92} C_VEL
LIN {X 0,Y 291.56,Z 319.162,A -85,B 0,C 180,E1 -16569.715,E2 -16569.715} C_VEL
LIN {X 0,Y 291.507,Z 319.16,A -85,B 0,C 180,E1 -16573.951,E2 -16573.951} C_VEL
LIN {X 0,Y 291.434,Z 319.165,A -85,B 0,C 180,E1 -16578.27,E2 -16578.27} C_VEL
LIN {X 0,Y 291.348,Z 319.19,A -85,B 0,C 180,E1 -16581.213,E2 -16581.213} C_VEL
LIN {X 0,Y 291.34,Z 319.188,A -85,B 0,C 180,E1 -16584.211,E2 -16584.211} C_VEL
LIN {X 0,Y 291.344,Z 319.184,A -85,B 0,C 180,E1 -16587.28,E2 -16587.28} C_VEL
LIN {X 0,Y 291.312,Z 319.196,A -85,B 0,C 180,E1 -16590.44,E2 -16590.44} C_VEL
LIN {X 0,Y 291.338,Z 319.196,A -85,B 0,C 180,E1 -16593.7,E2 -16593.7} C_VEL
LIN {X 0,Y 291.347,Z 319.195,A -85,B 0,C 180,E1 -16597.249,E2 -16597.249} C_VEL
LIN {X 0,Y 291.29,Z 319.194,A -85,B 0,C 180,E1 -16601.59,E2 -16601.59} C_VEL
LIN {X 0,Y 291.287,Z 319.202,A -85,B 0,C 180,E1 -16605.6,E2 -16605.6} C_VEL
LIN {X 0,Y 291.329,Z 319.198,A -85,B 0,C 180,E1 -16609.359,E2 -16609.359} C_VEL
LIN {X 0,Y 291.369,Z 319.223,A -85,B 0,C 180,E1 -16612.442,E2 -16612.442} C_VEL
LIN {X 0,Y 293.653,Z 327.779,A -85,B 0,C 180,E1 -16615.778,E2 -16615.778} C_VEL
LIN {X 0,Y 296.13,Z 338.185,A -85,B 0,C 180,E1 -16619.54,E2 -16619.54} C_VEL
LIN {X 0,Y 296.341,Z 339.054,A -85,B 0,C 180,E1 -16619.77,E2 -16619.77} C_VEL
LIN {X 0,Y 303.55,Z 354.626,A -85,B 0,C 180,E1 -16621.152,E2 -16621.152} C_VEL
LIN {X 0,Y 304.688,Z 358.378,A -85,B 0,C 180,E1 -16621.398,E2 -16621.398} C_VEL
LIN {X 0,Y 308.861,Z 380.221,A -85,B 0,C 180,E1 -16622.498,E2 -16622.498} C_VEL
LIN {X 0,Y 309.611,Z 385.716,A -85,B 0,C 180,E1 -16622.733,E2 -16622.733} C_VEL
LIN {X 0,Y 307.522,Z 447.945,A -85,B 0,C 180,E1 -16624.219,E2 -16624.219} C_VEL
LIN {X 0,Y 306.424,Z 461.68,A -85,B 0,C 180,E1 -16624.804,E2 -16624.804} C_VEL
LIN {X 0,Y 305.019,Z 472.94,A -85,B 0,C 180,E1 -16625.498,E2 -16625.498} C_VEL
LIN {X 0,Y 303.336,Z 484.294,A -85,B 0,C 180,E1 -16626.444,E2 -16626.444} C_VEL
LIN {X 0,Y 301.352,Z 495.972,A -85,B 0,C 180,E1 -16627.731,E2 -16627.731} C_VEL
LIN {X 0,Y 299.132,Z 506.479,A -85,B 0,C 180,E1 -16629.186,E2 -16629.186} C_VEL
LIN {X 0,Y 297.238,Z 515.077,A -85,B 0,C 180,E1 -16630.671,E2 -16630.671} C_VEL
LIN {X 0,Y 295.491,Z 523.014,A -85,B 0,C 180,E1 -16632.349,E2 -16632.349} C_VEL
LIN {X 0,Y 293.719,Z 530.826,A -85,B 0,C 180,E1 -16634.386,E2 -16634.386} C_VEL
LIN {X 0,Y 291.937,Z 538,A -85,B 0,C 180,E1 -16636.781,E2 -16636.781} C_VEL
LIN {X 0,Y 290.866,Z 542.819,A -85,B 0,C 180,E1 -16638.856,E2 -16638.856} C_VEL
LIN {X 0,Y 290.124,Z 546.542,A -85,B 0,C 180,E1 -16640.942,E2 -16640.942} C_VEL
LIN {X 0,Y 289.673,Z 549.269,A -85,B 0,C 180,E1 -16643.034,E2 -16643.034} C_VEL
LIN {X 0,Y 289.404,Z 551.48,A -85,B 0,C 180,E1 -16645.823,E2 -16645.823} C_VEL
LIN {X 0,Y 289.43,Z 551.975,A -85,B 0,C 180,E1 -16647.218,E2 -16647.218} C_VEL
LIN {X 0,Y 289.407,Z 552.06,A -85,B 0,C 180,E1 -16648.61,E2 -16648.61} C_VEL
LIN {X 0,Y 289.437,Z 551.761,A -85,B 0,C 180,E1 -16650.001,E2 -16650.001} C_VEL
LIN {X 0,Y 289.421,Z 551.072,A -85,B 0,C 180,E1 -16651.393,E2 -16651.393} C_VEL
LIN {X 0,Y 289.469,Z 549.967,A -85,B 0,C 180,E1 -16652.784,E2 -16652.784} C_VEL
LIN {X 0,Y 289.444,Z 548.409,A -85,B 0,C 180,E1 -16654.179,E2 -16654.179} C_VEL
LIN {X 0,Y 289.559,Z 545.271,A -85,B 0,C 180,E1 -16656.272,E2 -16656.272} C_VEL
LIN {X 0,Y 289.836,Z 541.05,A -85,B 0,C 180,E1 -16658.367,E2 -16658.367} C_VEL
LIN {X 0,Y 290.432,Z 534.604,A -85,B 0,C 180,E1 -16660.81,E2 -16660.81} C_VEL
LIN {X 0,Y 291.271,Z 527.555,A -85,B 0,C 180,E1 -16662.898,E2 -16662.898} C_VEL
LIN {X 0,Y 292.412,Z 518.698,A -85,B 0,C 180,E1 -16664.975,E2 -16664.975} C_VEL
LIN {X 0,Y 293.586,Z 509.608,A -85,B 0,C 180,E1 -16666.695,E2 -16666.695} C_VEL
LIN {X 0,Y 294.75,Z 499.577,A -85,B 0,C 180,E1 -16668.238,E2 -16668.238} C_VEL
LIN {X 0,Y 296.173,Z 488.45,A -85,B 0,C 180,E1 -16669.584,E2 -16669.584} C_VEL
LIN {X 0,Y 297.47,Z 475.942,A -85,B 0,C 180,E1 -16670.757,E2 -16670.757} C_VEL
LIN {X 0,Y 298.497,Z 464.031,A -85,B 0,C 180,E1 -16671.586,E2 -16671.586} C_VEL
LIN {X 0,Y 299.343,Z 451.047,A -85,B 0,C 180,E1 -16672.201,E2 -16672.201} C_VEL
LIN {X 0,Y 299.9,Z 432.818,A -85,B 0,C 180,E1 -16672.697,E2 -16672.697} C_VEL
LIN {X 0,Y 300.859,Z 380.577,A -85,B 0,C 180,E1 -16673.942,E2 -16673.942} C_VEL
LIN {X 0,Y 295.133,Z 339.711,A -85,B 0,C 180,E1 -16675.382,E2 -16675.382} C_VEL
LIN {X 0,Y 294.232,Z 333.045,A -85,B 0,C 180,E1 -16677.385,E2 -16677.385} C_VEL
LIN {X 0,Y 291.758,Z 320.968,A -85,B 0,C 180,E1 -16681.193,E2 -16681.193} C_VEL
LIN {X 0,Y 291.391,Z 319.183,A -85,B 0,C 180,E1 -16681.845,E2 -16681.845} C_VEL
LIN {X 0,Y 291.359,Z 319.191,A -85,B 0,C 180,E1 -16685.375,E2 -16685.375} C_VEL
LIN {X 0,Y 291.308,Z 319.197,A -85,B 0,C 180,E1 -16688.85,E2 -16688.85} C_VEL
LIN {X 0,Y 291.292,Z 319.202,A -85,B 0,C 180,E1 -16692.499,E2 -16692.499} C_VEL
LIN {X 0,Y 291.314,Z 319.2,A -85,B 0,C 180,E1 -16696.367,E2 -16696.367} C_VEL
LIN {X 0,Y 291.383,Z 319.192,A -85,B 0,C 180,E1 -16700.519,E2 -16700.519} C_VEL
LIN {X 0,Y 291.409,Z 319.187,A -85,B 0,C 180,E1 -16702.919,E2 -16702.919} C_VEL
LIN {X 0,Y 291.349,Z 319.191,A -85,B 0,C 180,E1 -16706.302,E2 -16706.302} C_VEL
LIN {X 0,Y 291.375,Z 319.187,A -85,B 0,C 180,E1 -16710.266,E2 -16710.266} C_VEL
LIN {X 0,Y 291.381,Z 319.186,A -85,B 0,C 180,E1 -16714.268,E2 -16714.268} C_VEL
LIN {X 0,Y 291.375,Z 319.189,A -85,B 0,C 180,E1 -16717.299,E2 -16717.299} C_VEL
LIN {X 0,Y 291.411,Z 319.175,A -85,B 0,C 180,E1 -16720.266,E2 -16720.266} C_VEL
LIN {X 0,Y 291.502,Z 319.171,A -85,B 0,C 180,E1 -16724.665,E2 -16724.665} C_VEL
LIN {X 0,Y 291.54,Z 319.162,A -85,B 0,C 180,E1 -16728.88,E2 -16728.88} C_VEL
LIN {X 0,Y 291.672,Z 319.145,A -85,B 0,C 180,E1 -16731.687,E2 -16731.687} C_VEL
LIN {X 0,Y 291.615,Z 319.157,A -85,B 0,C 180,E1 -16734.468,E2 -16734.468} C_VEL
LIN {X 0,Y 291.886,Z 319.122,A -85,B 0,C 180,E1 -16738.62,E2 -16738.62} C_VEL
LIN {X 0,Y 291.888,Z 319.116,A -85,B 0,C 180,E1 -16741.379,E2 -16741.379} C_VEL
LIN {X 0,Y 291.692,Z 319.148,A -85,B 0,C 180,E1 -16746.919,E2 -16746.919} C_VEL
LIN {X 0,Y 291.572,Z 319.162,A -85,B 0,C 180,E1 -16749.713,E2 -16749.713} C_VEL
LIN {X 0,Y 291.519,Z 319.163,A -85,B 0,C 180,E1 -16753.95,E2 -16753.95} C_VEL
LIN {X 0,Y 291.432,Z 319.176,A -85,B 0,C 180,E1 -16756.821,E2 -16756.821} C_VEL
LIN {X 0,Y 291.428,Z 319.179,A -85,B 0,C 180,E1 -16759.859,E2 -16759.859} C_VEL
LIN {X 0,Y 291.37,Z 319.185,A -85,B 0,C 180,E1 -16764.208,E2 -16764.208} C_VEL
LIN {X 0,Y 291.365,Z 319.182,A -85,B 0,C 180,E1 -16767.277,E2 -16767.277} C_VEL
LIN {X 0,Y 291.325,Z 319.189,A -85,B 0,C 180,E1 -16770.438,E2 -16770.438} C_VEL
LIN {X 0,Y 291.347,Z 319.192,A -85,B 0,C 180,E1 -16773.698,E2 -16773.698} C_VEL
LIN {X 0,Y 291.376,Z 319.185,A -85,B 0,C 180,E1 -16777.252,E2 -16777.252} C_VEL
LIN {X 0,Y 291.334,Z 319.189,A -85,B 0,C 180,E1 -16780.642,E2 -16780.642} C_VEL
LIN {X 0,Y 291.293,Z 319.197,A -85,B 0,C 180,E1 -16784.401,E2 -16784.401} C_VEL
LIN {X 0,Y 291.327,Z 319.192,A -85,B 0,C 180,E1 -16788.404,E2 -16788.404} C_VEL
LIN {X 0,Y 291.341,Z 319.191,A -85,B 0,C 180,E1 -16791.155,E2 -16791.155} C_VEL
LIN {X 0,Y 291.357,Z 319.187,A -85,B 0,C 180,E1 -16794.624,E2 -16794.624} C_VEL
LIN {X 0,Y 291.368,Z 319.19,A -85,B 0,C 180,E1 -16797.949,E2 -16797.949} C_VEL
LIN {X 0,Y 291.359,Z 319.189,A -85,B 0,C 180,E1 -16801.155,E2 -16801.155} C_VEL
LIN {X 0,Y 291.379,Z 319.189,A -85,B 0,C 180,E1 -16804.267,E2 -16804.267} C_VEL
LIN {X 0,Y 291.38,Z 319.188,A -85,B 0,C 180,E1 -16807.298,E2 -16807.298} C_VEL
LIN {X 0,Y 291.459,Z 319.179,A -85,B 0,C 180,E1 -16810.269,E2 -16810.269} C_VEL
LIN {X 0,Y 291.498,Z 319.176,A -85,B 0,C 180,E1 -16814.664,E2 -16814.664} C_VEL
LIN {X 0,Y 291.549,Z 319.275,A -85,B 0,C 180,E1 -16816.672,E2 -16816.672} C_VEL
LIN {X 0,Y 292.666,Z 324.747,A -85,B 0,C 180,E1 -16818.493,E2 -16818.493} C_VEL
LIN {X 0,Y 298.803,Z 342.72,A -85,B 0,C 180,E1 -16819.42,E2 -16819.42} C_VEL
LIN {X 0,Y 301.452,Z 358.095,A -85,B 0,C 180,E1 -16819.993,E2 -16819.993} C_VEL
LIN {X 0,Y 299.6,Z 432.662,A -85,B 0,C 180,E1 -16821.781,E2 -16821.781} C_VEL
LIN {X 0,Y 298.951,Z 444.916,A -85,B 0,C 180,E1 -16822.315,E2 -16822.315} C_VEL
LIN {X 0,Y 298.08,Z 457.686,A -85,B 0,C 180,E1 -16823.144,E2 -16823.144} C_VEL
LIN {X 0,Y 297.063,Z 469.105,A -85,B 0,C 180,E1 -16824.148,E2 -16824.148} C_VEL
LIN {X 0,Y 295.88,Z 480.106,A -85,B 0,C 180,E1 -16825.4,E2 -16825.4} C_VEL
LIN {X 0,Y 294.54,Z 490.741,A -85,B 0,C 180,E1 -16826.921,E2 -16826.921} C_VEL
LIN {X 0,Y 293.241,Z 500.327,A -85,B 0,C 180,E1 -16828.625,E2 -16828.625} C_VEL
LIN {X 0,Y 292.177,Z 508.167,A -85,B 0,C 180,E1 -16830.343,E2 -16830.343} C_VEL
LIN {X 0,Y 291.176,Z 515.817,A -85,B 0,C 180,E1 -16832.42,E2 -16832.42} C_VEL
LIN {X 0,Y 290.338,Z 522.882,A -85,B 0,C 180,E1 -16834.859,E2 -16834.859} C_VEL
LIN {X 0,Y 289.945,Z 527.563,A -85,B 0,C 180,E1 -16836.96,E2 -16836.96} C_VEL
LIN {X 0,Y 289.535,Z 531.149,A -85,B 0,C 180,E1 -16839.077,E2 -16839.077} C_VEL
LIN {X 0,Y 289.312,Z 533.706,A -85,B 0,C 180,E1 -16841.205,E2 -16841.205} C_VEL
LIN {X 0,Y 289.265,Z 535.454,A -85,B 0,C 180,E1 -16843.63,E2 -16843.63} C_VEL
LIN {X 0,Y 289.26,Z 535.948,A -85,B 0,C 180,E1 -16845.5,E2 -16845.5} C_VEL
LIN {X 0,Y 289.358,Z 535.884,A -85,B 0,C 180,E1 -16846.944,E2 -16846.944} C_VEL
LIN {X 0,Y 289.69,Z 535.079,A -85,B 0,C 180,E1 -16848.888,E2 -16848.888} C_VEL
LIN {X 0,Y 290.19,Z 533.045,A -85,B 0,C 180,E1 -16851.3,E2 -16851.3} C_VEL
LIN {X 0,Y 290.947,Z 530.263,A -85,B 0,C 180,E1 -16853.378,E2 -16853.378} C_VEL
LIN {X 0,Y 291.982,Z 526.036,A -85,B 0,C 180,E1 -16855.673,E2 -16855.673} C_VEL
LIN {X 0,Y 293.419,Z 520.425,A -85,B 0,C 180,E1 -16857.942,E2 -16857.942} C_VEL
LIN {X 0,Y 295.064,Z 513.873,A -85,B 0,C 180,E1 -16860.011,E2 -16860.011} C_VEL
LIN {X 0,Y 297.104,Z 505.305,A -85,B 0,C 180,E1 -16862.155,E2 -16862.155} C_VEL
LIN {X 0,Y 299.128,Z 496.409,A -85,B 0,C 180,E1 -16863.916,E2 -16863.916} C_VEL
LIN {X 0,Y 301.099,Z 486.768,A -85,B 0,C 180,E1 -16865.45,E2 -16865.45} C_VEL
LIN {X 0,Y 303.122,Z 475.632,A -85,B 0,C 180,E1 -16866.862,E2 -16866.862} C_VEL
LIN {X 0,Y 304.673,Z 465.408,A -85,B 0,C 180,E1 -16867.89,E2 -16867.89} C_VEL
LIN {X 0,Y 306.255,Z 452.871,A -85,B 0,C 180,E1 -16868.847,E2 -16868.847} C_VEL
LIN {X 0,Y 307.338,Z 439.885,A -85,B 0,C 180,E1 -16869.553,E2 -16869.553} C_VEL
LIN {X 0,Y 308.079,Z 427.215,A -85,B 0,C 180,E1 -16869.979,E2 -16869.979} C_VEL
LIN {X 0,Y 310.317,Z 361.569,A -85,B 0,C 180,E1 -16871.502,E2 -16871.502} C_VEL
LIN {X 0,Y 305.121,Z 349.205,A -85,B 0,C 180,E1 -16872.467,E2 -16872.467} C_VEL
LIN {X 0,Y 297.308,Z 333.446,A -85,B 0,C 180,E1 -16873.926,E2 -16873.926} C_VEL
LIN {X 0,Y 292.933,Z 325.312,A -85,B 0,C 180,E1 -16874.776,E2 -16874.776} C_VEL
LIN {X 0,Y 291.303,Z 319.187,A -85,B 0,C 180,E1 -16877.246,E2 -16877.246} C_VEL
LIN {X 0,Y 291.328,Z 319.2,A -85,B 0,C 180,E1 -16881.155,E2 -16881.155} C_VEL
LIN {X 0,Y 291.353,Z 319.182,A -85,B 0,C 180,E1 -16884.625,E2 -16884.625} C_VEL
LIN {X 0,Y 291.32,Z 319.173,A -85,B 0,C 180,E1 -16886.651,E2 -16886.651} C_VEL
LIN {X 0,Y 290.624,Z 319.274,A -85,B 0,C 180,E1 -16887.806,E2 -16887.806} C_VEL
LIN {X 0,Y 287.736,Z 319.641,A -85,B 0,C 180,E1 -16889.685,E2 -16889.685} C_VEL
LIN {X 0,Y 285.338,Z 319.941,A -85,B 0,C 180,E1 -16891.212,E2 -16891.212} C_VEL
LIN {X 0,Y 284.364,Z 320.064,A -85,B 0,C 180,E1 -16892.395,E2 -16892.395} C_VEL
LIN {X 0,Y 284.313,Z 320.07,A -85,B 0,C 180,E1 -16892.795,E2 -16892.795} C_VEL
LIN {X 0,Y 284.311,Z 320.068,A -85,B 0,C 180,E1 -16896.703,E2 -16896.703} C_VEL
LIN {X 0,Y 284.314,Z 320.063,A -85,B 0,C 180,E1 -16901.256,E2 -16901.256} C_VEL
LIN {X 0,Y 284.409,Z 320.049,A -85,B 0,C 180,E1 -16905.694,E2 -16905.694} C_VEL
LIN {X 0,Y 284.505,Z 320.039,A -85,B 0,C 180,E1 -16910.043,E2 -16910.043} C_VEL
LIN {X 0,Y 284.631,Z 320.024,A -85,B 0,C 180,E1 -16912.909,E2 -16912.909} C_VEL
LIN {X 0,Y 284.824,Z 320.003,A -85,B 0,C 180,E1 -16918.586,E2 -16918.586} C_VEL
LIN {X 0,Y 284.834,Z 319.993,A -85,B 0,C 180,E1 -16921.414,E2 -16921.414} C_VEL
LIN {X 0,Y 284.638,Z 320.014,A -85,B 0,C 180,E1 -16927.092,E2 -16927.092} C_VEL
LIN {X 0,Y 284.506,Z 320.041,A -85,B 0,C 180,E1 -16929.958,E2 -16929.958} C_VEL
LIN {X 0,Y 284.455,Z 320.04,A -85,B 0,C 180,E1 -16934.304,E2 -16934.304} C_VEL
LIN {X 0,Y 284.374,Z 320.046,A -85,B 0,C 180,E1 -16938.741,E2 -16938.741} C_VEL
LIN {X 0,Y 284.301,Z 320.064,A -85,B 0,C 180,E1 -16941.766,E2 -16941.766} C_VEL
LIN {X 0,Y 284.288,Z 320.069,A -85,B 0,C 180,E1 -16944.852,E2 -16944.852} C_VEL
LIN {X 0,Y 284.275,Z 320.065,A -85,B 0,C 180,E1 -16948.017,E2 -16948.017} C_VEL
LIN {X 0,Y 284.279,Z 320.066,A -85,B 0,C 180,E1 -16951.277,E2 -16951.277} C_VEL
LIN {X 0,Y 284.331,Z 320.06,A -85,B 0,C 180,E1 -16955.348,E2 -16955.348} C_VEL
LIN {X 0,Y 284.258,Z 320.073,A -85,B 0,C 180,E1 -16958.178,E2 -16958.178} C_VEL
LIN {X 0,Y 284.232,Z 320.066,A -85,B 0,C 180,E1 -16962.119,E2 -16962.119} C_VEL
LIN {X 0,Y 284.252,Z 320.084,A -85,B 0,C 180,E1 -16966.191,E2 -16966.191} C_VEL
LIN {X 0,Y 284.303,Z 320.073,A -85,B 0,C 180,E1 -16970.025,E2 -16970.025} C_VEL
LIN {X 0,Y 284.347,Z 320.268,A -85,B 0,C 180,E1 -16971.613,E2 -16971.613} C_VEL
LIN {X 0,Y 286.529,Z 328.286,A -85,B 0,C 180,E1 -16974.877,E2 -16974.877} C_VEL
LIN {X 0,Y 289.047,Z 338.631,A -85,B 0,C 180,E1 -16978.743,E2 -16978.743} C_VEL
LIN {X 0,Y 297.055,Z 355.5,A -85,B 0,C 180,E1 -16980.346,E2 -16980.346} C_VEL
LIN {X 0,Y 298.842,Z 360.17,A -85,B 0,C 180,E1 -16980.713,E2 -16980.713} C_VEL
LIN {X 0,Y 303.011,Z 382.36,A -85,B 0,C 180,E1 -16981.863,E2 -16981.863} C_VEL
LIN {X 0,Y 303.553,Z 386.732,A -85,B 0,C 180,E1 -16982.05,E2 -16982.05} C_VEL
LIN {X 0,Y 301.41,Z 448.029,A -85,B 0,C 180,E1 -16983.544,E2 -16983.544} C_VEL
LIN {X 0,Y 300.228,Z 461.976,A -85,B 0,C 180,E1 -16984.153,E2 -16984.153} C_VEL
LIN {X 0,Y 298.623,Z 474.19,A -85,B 0,C 180,E1 -16984.938,E2 -16984.938} C_VEL
LIN {X 0,Y 296.66,Z 486.715,A -85,B 0,C 180,E1 -16986.067,E2 -16986.067} C_VEL
LIN {X 0,Y 294.533,Z 497.896,A -85,B 0,C 180,E1 -16987.372,E2 -16987.372} C_VEL
LIN {X 0,Y 292.323,Z 508.004,A -85,B 0,C 180,E1 -16988.863,E2 -16988.863} C_VEL
LIN {X 0,Y 290.165,Z 517.122,A -85,B 0,C 180,E1 -16990.549,E2 -16990.549} C_VEL
LIN {X 0,Y 288.38,Z 524.818,A -85,B 0,C 180,E1 -16992.307,E2 -16992.307} C_VEL
LIN {X 0,Y 286.587,Z 532.093,A -85,B 0,C 180,E1 -16994.352,E2 -16994.352} C_VEL
LIN {X 0,Y 285.023,Z 538.085,A -85,B 0,C 180,E1 -16996.454,E2 -16996.454} C_VEL
LIN {X 0,Y 283.89,Z 542.844,A -85,B 0,C 180,E1 -16998.579,E2 -16998.579} C_VEL
LIN {X 0,Y 283.099,Z 546.51,A -85,B 0,C 180,E1 -17000.715,E2 -17000.715} C_VEL
LIN {X 0,Y 282.604,Z 549.184,A -85,B 0,C 180,E1 -17002.858,E2 -17002.858} C_VEL
LIN {X 0,Y 282.397,Z 550.665,A -85,B 0,C 180,E1 -17004.554,E2 -17004.554} C_VEL
LIN {X 0,Y 282.337,Z 551.788,A -85,B 0,C 180,E1 -17007.148,E2 -17007.148} C_VEL
LIN {X 0,Y 282.331,Z 551.849,A -85,B 0,C 180,E1 -17008.575,E2 -17008.575} C_VEL
LIN {X 0,Y 282.357,Z 551.524,A -85,B 0,C 180,E1 -17010.001,E2 -17010.001} C_VEL
LIN {X 0,Y 282.345,Z 550.81,A -85,B 0,C 180,E1 -17011.428,E2 -17011.428} C_VEL
LIN {X 0,Y 282.374,Z 549.653,A -85,B 0,C 180,E1 -17012.855,E2 -17012.855} C_VEL
LIN {X 0,Y 282.411,Z 546.422,A -85,B 0,C 180,E1 -17015.476,E2 -17015.476} C_VEL
LIN {X 0,Y 282.67,Z 542.156,A -85,B 0,C 180,E1 -17017.861,E2 -17017.861} C_VEL
LIN {X 0,Y 283.098,Z 537.093,A -85,B 0,C 180,E1 -17020.009,E2 -17020.009} C_VEL
LIN {X 0,Y 283.791,Z 530.709,A -85,B 0,C 180,E1 -17022.153,E2 -17022.153} C_VEL
LIN {X 0,Y 284.911,Z 522.7,A -85,B 0,C 180,E1 -17024.282,E2 -17024.282} C_VEL
LIN {X 0,Y 286.235,Z 513.174,A -85,B 0,C 180,E1 -17026.309,E2 -17026.309} C_VEL
LIN {X 0,Y 287.37,Z 503.383,A -85,B 0,C 180,E1 -17027.986,E2 -17027.986} C_VEL
LIN {X 0,Y 288.679,Z 493.234,A -85,B 0,C 180,E1 -17029.374,E2 -17029.374} C_VEL
LIN {X 0,Y 290.027,Z 482.182,A -85,B 0,C 180,E1 -17030.572,E2 -17030.572} C_VEL
LIN {X 0,Y 291.249,Z 469.931,A -85,B 0,C 180,E1 -17031.593,E2 -17031.593} C_VEL
LIN {X 0,Y 292.187,Z 457.119,A -85,B 0,C 180,E1 -17032.356,E2 -17032.356} C_VEL
LIN {X 0,Y 292.871,Z 443.205,A -85,B 0,C 180,E1 -17032.872,E2 -17032.872} C_VEL
LIN {X 0,Y 294.168,Z 381.406,A -85,B 0,C 180,E1 -17034.377,E2 -17034.377} C_VEL
LIN {X 0,Y 288.625,Z 341.609,A -85,B 0,C 180,E1 -17035.817,E2 -17035.817} C_VEL
LIN {X 0,Y 288.117,Z 339.465,A -85,B 0,C 180,E1 -17035.926,E2 -17035.926} C_VEL
LIN {X 0,Y 286.34,Z 329.542,A -85,B 0,C 180,E1 -17039.045,E2 -17039.045} C_VEL
LIN {X 0,Y 284.334,Z 320.06,A -85,B 0,C 180,E1 -17042.191,E2 -17042.191} C_VEL
LIN {X 0,Y 284.323,Z 320.069,A -85,B 0,C 180,E1 -17046.389,E2 -17046.389} C_VEL
LIN {X 0,Y 284.259,Z 320.078,A -85,B 0,C 180,E1 -17050.004,E2 -17050.004} C_VEL
LIN {X 0,Y 284.239,Z 320.082,A -85,B 0,C 180,E1 -17054.188,E2 -17054.188} C_VEL
LIN {X 0,Y 284.277,Z 320.075,A -85,B 0,C 180,E1 -17058.125,E2 -17058.125} C_VEL
LIN {X 0,Y 284.324,Z 320.067,A -85,B 0,C 180,E1 -17062.279,E2 -17062.279} C_VEL
LIN {X 0,Y 284.313,Z 320.067,A -85,B 0,C 180,E1 -17065.351,E2 -17065.351} C_VEL
LIN {X 0,Y 284.291,Z 320.073,A -85,B 0,C 180,E1 -17068.725,E2 -17068.725} C_VEL
LIN {X 0,Y 284.296,Z 320.068,A -85,B 0,C 180,E1 -17071.985,E2 -17071.985} C_VEL
LIN {X 0,Y 284.33,Z 320.064,A -85,B 0,C 180,E1 -17076.145,E2 -17076.145} C_VEL
LIN {X 0,Y 284.381,Z 320.051,A -85,B 0,C 180,E1 -17079.904,E2 -17079.904} C_VEL
LIN {X 0,Y 284.451,Z 320.049,A -85,B 0,C 180,E1 -17084.493,E2 -17084.493} C_VEL
LIN {X 0,Y 284.492,Z 320.04,A -85,B 0,C 180,E1 -17088.601,E2 -17088.601} C_VEL
LIN {X 0,Y 284.626,Z 320.019,A -85,B 0,C 180,E1 -17091.48,E2 -17091.48} C_VEL
LIN {X 0,Y 284.585,Z 320.033,A -85,B 0,C 180,E1 -17094.331,E2 -17094.331} C_VEL
LIN {X 0,Y 284.852,Z 319.998,A -85,B 0,C 180,E1 -17098.586,E2 -17098.586} C_VEL
LIN {X 0,Y 284.854,Z 319.992,A -85,B 0,C 180,E1 -17101.413,E2 -17101.413} C_VEL
LIN {X 0,Y 284.647,Z 320.025,A -85,B 0,C 180,E1 -17107.091,E2 -17107.091} C_VEL
LIN {X 0,Y 284.518,Z 320.042,A -85,B 0,C 180,E1 -17109.957,E2 -17109.957} C_VEL
LIN {X 0,Y 284.467,Z 320.042,A -85,B 0,C 180,E1 -17114.303,E2 -17114.303} C_VEL
LIN {X 0,Y 284.344,Z 320.063,A -85,B 0,C 180,E1 -17118.742,E2 -17118.742} C_VEL
LIN {X 0,Y 284.316,Z 320.066,A -85,B 0,C 180,E1 -17121.764,E2 -17121.764} C_VEL
LIN {X 0,Y 284.319,Z 320.067,A -85,B 0,C 180,E1 -17124.848,E2 -17124.848} C_VEL
LIN {X 0,Y 284.294,Z 320.058,A -85,B 0,C 180,E1 -17128.014,E2 -17128.014} C_VEL
LIN {X 0,Y 284.29,Z 320.07,A -85,B 0,C 180,E1 -17131.275,E2 -17131.275} C_VEL
LIN {X 0,Y 284.344,Z 320.065,A -85,B 0,C 180,E1 -17135.347,E2 -17135.347} C_VEL
LIN {X 0,Y 284.311,Z 320.057,A -85,B 0,C 180,E1 -17138.169,E2 -17138.169} C_VEL
LIN {X 0,Y 284.271,Z 320.073,A -85,B 0,C 180,E1 -17142.123,E2 -17142.123} C_VEL
LIN {X 0,Y 284.258,Z 320.07,A -85,B 0,C 180,E1 -17146.188,E2 -17146.188} C_VEL
LIN {X 0,Y 284.308,Z 320.07,A -85,B 0,C 180,E1 -17150.023,E2 -17150.023} C_VEL
LIN {X 0,Y 284.323,Z 320.066,A -85,B 0,C 180,E1 -17153.611,E2 -17153.611} C_VEL
LIN {X 0,Y 284.308,Z 320.067,A -85,B 0,C 180,E1 -17157.189,E2 -17157.189} C_VEL
LIN {X 0,Y 284.347,Z 320.067,A -85,B 0,C 180,E1 -17160.373,E2 -17160.373} C_VEL
LIN {X 0,Y 284.327,Z 320.065,A -85,B 0,C 180,E1 -17163.58,E2 -17163.58} C_VEL
LIN {X 0,Y 284.335,Z 320.07,A -85,B 0,C 180,E1 -17166.703,E2 -17166.703} C_VEL
LIN {X 0,Y 284.389,Z 320.059,A -85,B 0,C 180,E1 -17169.897,E2 -17169.897} C_VEL
LIN {X 0,Y 284.448,Z 320.053,A -85,B 0,C 180,E1 -17174.491,E2 -17174.491} C_VEL
LIN {X 0,Y 284.533,Z 320.249,A -85,B 0,C 180,E1 -17176.337,E2 -17176.337} C_VEL
LIN {X 0,Y 285.5,Z 324.95,A -85,B 0,C 180,E1 -17177.947,E2 -17177.947} C_VEL
LIN {X 0,Y 292.312,Z 344.578,A -85,B 0,C 180,E1 -17178.996,E2 -17178.996} C_VEL
LIN {X 0,Y 294.767,Z 358.117,A -85,B 0,C 180,E1 -17179.526,E2 -17179.526} C_VEL
LIN {X 0,Y 292.875,Z 432.184,A -85,B 0,C 180,E1 -17181.332,E2 -17181.332} C_VEL
LIN {X 0,Y 292.179,Z 445.379,A -85,B 0,C 180,E1 -17181.918,E2 -17181.918} C_VEL
LIN {X 0,Y 291.222,Z 458.645,A -85,B 0,C 180,E1 -17182.807,E2 -17182.807} C_VEL
LIN {X 0,Y 290.071,Z 471.141,A -85,B 0,C 180,E1 -17183.976,E2 -17183.976} C_VEL
LIN {X 0,Y 288.638,Z 483.329,A -85,B 0,C 180,E1 -17185.46,E2 -17185.46} C_VEL
LIN {X 0,Y 287.46,Z 492.367,A -85,B 0,C 180,E1 -17186.845,E2 -17186.845} C_VEL
LIN {X 0,Y 286.125,Z 501.646,A -85,B 0,C 180,E1 -17188.591,E2 -17188.591} C_VEL
LIN {X 0,Y 284.835,Z 510.648,A -85,B 0,C 180,E1 -17190.706,E2 -17190.706} C_VEL
LIN {X 0,Y 283.886,Z 517.893,A -85,B 0,C 180,E1 -17192.837,E2 -17192.837} C_VEL
LIN {X 0,Y 283.236,Z 523.669,A -85,B 0,C 180,E1 -17194.981,E2 -17194.981} C_VEL
LIN {X 0,Y 282.804,Z 528.216,A -85,B 0,C 180,E1 -17197.136,E2 -17197.136} C_VEL
LIN {X 0,Y 282.538,Z 530.623,A -85,B 0,C 180,E1 -17198.582,E2 -17198.582} C_VEL
LIN {X 0,Y 282.329,Z 532.599,A -85,B 0,C 180,E1 -17200.034,E2 -17200.034} C_VEL
LIN {X 0,Y 282.196,Z 534.142,A -85,B 0,C 180,E1 -17201.491,E2 -17201.491} C_VEL
LIN {X 0,Y 282.161,Z 535.655,A -85,B 0,C 180,E1 -17203.736,E2 -17203.736} C_VEL
LIN {X 0,Y 282.174,Z 536.18,A -85,B 0,C 180,E1 -17205.899,E2 -17205.899} C_VEL
LIN {X 0,Y 282.322,Z 536.018,A -85,B 0,C 180,E1 -17207.379,E2 -17207.379} C_VEL
LIN {X 0,Y 282.639,Z 535.287,A -85,B 0,C 180,E1 -17209.111,E2 -17209.111} C_VEL
LIN {X 0,Y 283.261,Z 532.976,A -85,B 0,C 180,E1 -17211.848,E2 -17211.848} C_VEL
LIN {X 0,Y 283.97,Z 530.51,A -85,B 0,C 180,E1 -17213.693,E2 -17213.693} C_VEL
LIN {X 0,Y 285.262,Z 525.691,A -85,B 0,C 180,E1 -17216.324,E2 -17216.324} C_VEL
LIN {X 0,Y 286.986,Z 519.241,A -85,B 0,C 180,E1 -17218.883,E2 -17218.883} C_VEL
LIN {X 0,Y 288.909,Z 512.143,A -85,B 0,C 180,E1 -17221.054,E2 -17221.054} C_VEL
LIN {X 0,Y 290.748,Z 504.409,A -85,B 0,C 180,E1 -17222.946,E2 -17222.946} C_VEL
LIN {X 0,Y 292.943,Z 495.251,A -85,B 0,C 180,E1 -17224.734,E2 -17224.734} C_VEL
LIN {X 0,Y 295.008,Z 485.623,A -85,B 0,C 180,E1 -17226.25,E2 -17226.25} C_VEL
LIN {X 0,Y 296.909,Z 475.361,A -85,B 0,C 180,E1 -17227.553,E2 -17227.553} C_VEL
LIN {X 0,Y 298.657,Z 464.039,A -85,B 0,C 180,E1 -17228.685,E2 -17228.685} C_VEL
LIN {X 0,Y 300.228,Z 451.878,A -85,B 0,C 180,E1 -17229.589,E2 -17229.589} C_VEL
LIN {X 0,Y 301.314,Z 439.051,A -85,B 0,C 180,E1 -17230.278,E2 -17230.278} C_VEL
LIN {X 0,Y 302.06,Z 425.887,A -85,B 0,C 180,E1 -17230.702,E2 -17230.702} C_VEL
LIN {X 0,Y 304.247,Z 363.162,A -85,B 0,C 180,E1 -17232.185,E2 -17232.185} C_VEL
LIN {X 0,Y 298.034,Z 349.015,A -85,B 0,C 180,E1 -17233.376,E2 -17233.376} C_VEL
LIN {X 0,Y 289.767,Z 332.947,A -85,B 0,C 180,E1 -17234.989,E2 -17234.989} C_VEL
LIN {X 0,Y 285.749,Z 325.552,A -85,B 0,C 180,E1 -17235.82,E2 -17235.82} C_VEL
LIN {X 0,Y 284.247,Z 320.07,A -85,B 0,C 180,E1 -17238.12,E2 -17238.12} C_VEL
LIN {X 0,Y 284.307,Z 320.068,A -85,B 0,C 180,E1 -17242.279,E2 -17242.279} C_VEL
LIN {X 0,Y 284.301,Z 320.05,A -85,B 0,C 180,E1 -17245.35,E2 -17245.35} C_VEL
LIN {X 0,Y 284.277,Z 320.075,A -85,B 0,C 180,E1 -17248.724,E2 -17248.724} C_VEL
LIN {X 0,Y 284.273,Z 320.076,A -85,B 0,C 180,E1 -17251.984,E2 -17251.984} C_VEL
LIN {X 0,Y 284.313,Z 320.07,A -85,B 0,C 180,E1 -17252.795,E2 -17252.795} C_VEL
LIN {X 0,Y 284.046,Z 320.105,A -85,B 0,C 180,E1 -17253.586,E2 -17253.586} C_VEL
LIN {X 0,Y 282.713,Z 320.273,A -85,B 0,C 180,E1 -17254.752,E2 -17254.752} C_VEL
LIN {X 0,Y 278.334,Z 320.807,A -85,B 0,C 180,E1 -17257.462,E2 -17257.462} C_VEL
LIN {X 0,Y 277.307,Z 320.936,A -85,B 0,C 180,E1 -17258.675,E2 -17258.675} C_VEL
LIN {X 0,Y 277.245,Z 320.946,A -85,B 0,C 180,E1 -17259.086,E2 -17259.086} C_VEL
LIN {X 0,Y 277.283,Z 320.934,A -85,B 0,C 180,E1 -17262.293,E2 -17262.293} C_VEL
LIN {X 0,Y 277.362,Z 320.931,A -85,B 0,C 180,E1 -17265.322,E2 -17265.322} C_VEL
LIN {X 0,Y 277.444,Z 320.922,A -85,B 0,C 180,E1 -17269.787,E2 -17269.787} C_VEL
LIN {X 0,Y 277.59,Z 320.898,A -85,B 0,C 180,E1 -17272.728,E2 -17272.728} C_VEL
LIN {X 0,Y 277.789,Z 320.878,A -85,B 0,C 180,E1 -17278.551,E2 -17278.551} C_VEL
LIN {X 0,Y 277.8,Z 320.869,A -85,B 0,C 180,E1 -17281.45,E2 -17281.45} C_VEL
LIN {X 0,Y 277.596,Z 320.889,A -85,B 0,C 180,E1 -17287.273,E2 -17287.273} C_VEL
LIN {X 0,Y 277.449,Z 320.921,A -85,B 0,C 180,E1 -17290.214,E2 -17290.214} C_VEL
LIN {X 0,Y 277.402,Z 320.921,A -85,B 0,C 180,E1 -17294.676,E2 -17294.676} C_VEL
LIN {X 0,Y 277.321,Z 320.927,A -85,B 0,C 180,E1 -17299.236,E2 -17299.236} C_VEL
LIN {X 0,Y 277.265,Z 320.938,A -85,B 0,C 180,E1 -17303.927,E2 -17303.927} C_VEL
LIN {X 0,Y 277.261,Z 320.937,A -85,B 0,C 180,E1 -17307.483,E2 -17307.483} C_VEL
LIN {X 0,Y 277.242,Z 320.949,A -85,B 0,C 180,E1 -17310.474,E2 -17310.474} C_VEL
LIN {X 0,Y 277.24,Z 320.951,A -85,B 0,C 180,E1 -17313.897,E2 -17313.897} C_VEL
LIN {X 0,Y 277.227,Z 320.954,A -85,B 0,C 180,E1 -17317.476,E2 -17317.476} C_VEL
LIN {X 0,Y 277.172,Z 320.957,A -85,B 0,C 180,E1 -17321.244,E2 -17321.244} C_VEL
LIN {X 0,Y 277.194,Z 320.949,A -85,B 0,C 180,E1 -17325.229,E2 -17325.229} C_VEL
LIN {X 0,Y 277.219,Z 320.955,A -85,B 0,C 180,E1 -17329.514,E2 -17329.514} C_VEL
LIN {X 0,Y 277.299,Z 321.073,A -85,B 0,C 180,E1 -17330.63,E2 -17330.63} C_VEL
LIN {X 0,Y 279.509,Z 329.02,A -85,B 0,C 180,E1 -17334.011,E2 -17334.011} C_VEL
LIN {X 0,Y 281.729,Z 338.27,A -85,B 0,C 180,E1 -17337.635,E2 -17337.635} C_VEL
LIN {X 0,Y 290.247,Z 355.64,A -85,B 0,C 180,E1 -17339.428,E2 -17339.428} C_VEL
LIN {X 0,Y 293.217,Z 362.924,A -85,B 0,C 180,E1 -17340.053,E2 -17340.053} C_VEL
LIN {X 0,Y 297.201,Z 384.475,A -85,B 0,C 180,E1 -17341.202,E2 -17341.202} C_VEL
LIN {X 0,Y 297.515,Z 388.726,A -85,B 0,C 180,E1 -17341.364,E2 -17341.364} C_VEL
LIN {X 0,Y 295.34,Z 447.607,A -85,B 0,C 180,E1 -17342.819,E2 -17342.819} C_VEL
LIN {X 0,Y 294.258,Z 460.759,A -85,B 0,C 180,E1 -17343.398,E2 -17343.398} C_VEL
LIN {X 0,Y 292.577,Z 473.272,A -85,B 0,C 180,E1 -17344.192,E2 -17344.192} C_VEL
LIN {X 0,Y 290.787,Z 484.422,A -85,B 0,C 180,E1 -17345.171,E2 -17345.171} C_VEL
LIN {X 0,Y 288.553,Z 495.985,A -85,B 0,C 180,E1 -17346.497,E2 -17346.497} C_VEL
LIN {X 0,Y 286.249,Z 506.407,A -85,B 0,C 180,E1 -17348.013,E2 -17348.013} C_VEL
LIN {X 0,Y 283.921,Z 515.827,A -85,B 0,C 180,E1 -17349.725,E2 -17349.725} C_VEL
LIN {X 0,Y 282.038,Z 523.379,A -85,B 0,C 180,E1 -17351.428,E2 -17351.428} C_VEL
LIN {X 0,Y 280.088,Z 531.143,A -85,B 0,C 180,E1 -17353.605,E2 -17353.605} C_VEL
LIN {X 0,Y 278.097,Z 538.177,A -85,B 0,C 180,E1 -17356.11,E2 -17356.11} C_VEL
LIN {X 0,Y 276.929,Z 542.87,A -85,B 0,C 180,E1 -17358.287,E2 -17358.287} C_VEL
LIN {X 0,Y 276.089,Z 546.477,A -85,B 0,C 180,E1 -17360.477,E2 -17360.477} C_VEL
LIN {X 0,Y 275.532,Z 549.098,A -85,B 0,C 180,E1 -17362.674,E2 -17362.674} C_VEL
LIN {X 0,Y 275.312,Z 550.645,A -85,B 0,C 180,E1 -17364.608,E2 -17364.608} C_VEL
LIN {X 0,Y 275.246,Z 551.602,A -85,B 0,C 180,E1 -17367.074,E2 -17367.074} C_VEL
LIN {X 0,Y 275.255,Z 551.637,A -85,B 0,C 180,E1 -17368.538,E2 -17368.538} C_VEL
LIN {X 0,Y 275.278,Z 551.288,A -85,B 0,C 180,E1 -17370.001,E2 -17370.001} C_VEL
LIN {X 0,Y 275.27,Z 550.536,A -85,B 0,C 180,E1 -17371.464,E2 -17371.464} C_VEL
LIN {X 0,Y 275.282,Z 549.339,A -85,B 0,C 180,E1 -17372.928,E2 -17372.928} C_VEL
LIN {X 0,Y 275.321,Z 546.354,A -85,B 0,C 180,E1 -17375.412,E2 -17375.412} C_VEL
LIN {X 0,Y 275.595,Z 541.729,A -85,B 0,C 180,E1 -17378.064,E2 -17378.064} C_VEL
LIN {X 0,Y 276.167,Z 535.601,A -85,B 0,C 180,E1 -17380.633,E2 -17380.633} C_VEL
LIN {X 0,Y 276.97,Z 528.874,A -85,B 0,C 180,E1 -17382.829,E2 -17382.829} C_VEL
LIN {X 0,Y 278.138,Z 520.514,A -85,B 0,C 180,E1 -17385.012,E2 -17385.012} C_VEL
LIN {X 0,Y 279.306,Z 512.857,A -85,B 0,C 180,E1 -17386.631,E2 -17386.631} C_VEL
LIN {X 0,Y 280.418,Z 503.607,A -85,B 0,C 180,E1 -17388.258,E2 -17388.258} C_VEL
LIN {X 0,Y 281.757,Z 493.561,A -85,B 0,C 180,E1 -17389.679,E2 -17389.679} C_VEL
LIN {X 0,Y 283.151,Z 482.637,A -85,B 0,C 180,E1 -17390.905,E2 -17390.905} C_VEL
LIN {X 0,Y 284.393,Z 470.563,A -85,B 0,C 180,E1 -17391.95,E2 -17391.95} C_VEL
LIN {X 0,Y 285.423,Z 457.345,A -85,B 0,C 180,E1 -17392.772,E2 -17392.772} C_VEL
LIN {X 0,Y 286.125,Z 443.806,A -85,B 0,C 180,E1 -17393.296,E2 -17393.296} C_VEL
LIN {X 0,Y 287.491,Z 382.282,A -85,B 0,C 180,E1 -17394.83,E2 -17394.83} C_VEL
LIN {X 0,Y 282.156,Z 343.437,A -85,B 0,C 180,E1 -17396.272,E2 -17396.272} C_VEL
LIN {X 0,Y 280.933,Z 339.217,A -85,B 0,C 180,E1 -17396.511,E2 -17396.511} C_VEL
LIN {X 0,Y 278.991,Z 328.977,A -85,B 0,C 180,E1 -17399.837,E2 -17399.837} C_VEL
LIN {X 0,Y 277.287,Z 320.938,A -85,B 0,C 180,E1 -17402.611,E2 -17402.611} C_VEL
LIN {X 0,Y 277.277,Z 320.945,A -85,B 0,C 180,E1 -17405.797,E2 -17405.797} C_VEL
LIN {X 0,Y 277.194,Z 320.955,A -85,B 0,C 180,E1 -17409.336,E2 -17409.336} C_VEL
LIN {X 0,Y 277.196,Z 320.955,A -85,B 0,C 180,E1 -17413.202,E2 -17413.202} C_VEL
LIN {X 0,Y 277.22,Z 320.953,A -85,B 0,C 180,E1 -17417.326,E2 -17417.326} C_VEL
LIN {X 0,Y 277.266,Z 320.944,A -85,B 0,C 180,E1 -17421.794,E2 -17421.794} C_VEL
LIN {X 0,Y 277.289,Z 320.944,A -85,B 0,C 180,E1 -17424.342,E2 -17424.342} C_VEL
LIN {X 0,Y 277.245,Z 320.947,A -85,B 0,C 180,E1 -17427.836,E2 -17427.836} C_VEL
LIN {X 0,Y 277.25,Z 320.95,A -85,B 0,C 180,E1 -17431.208,E2 -17431.208} C_VEL
LIN {X 0,Y 277.264,Z 320.945,A -85,B 0,C 180,E1 -17434.474,E2 -17434.474} C_VEL
LIN {X 0,Y 277.268,Z 320.942,A -85,B 0,C 180,E1 -17437.653,E2 -17437.653} C_VEL
LIN {X 0,Y 277.309,Z 320.931,A -85,B 0,C 180,E1 -17440.763,E2 -17440.763} C_VEL
LIN {X 0,Y 277.414,Z 320.929,A -85,B 0,C 180,E1 -17445.324,E2 -17445.324} C_VEL
LIN {X 0,Y 277.465,Z 320.912,A -85,B 0,C 180,E1 -17449.787,E2 -17449.787} C_VEL
LIN {X 0,Y 277.621,Z 320.895,A -85,B 0,C 180,E1 -17452.728,E2 -17452.728} C_VEL
LIN {X 0,Y 277.818,Z 320.874,A -85,B 0,C 180,E1 -17458.55,E2 -17458.55} C_VEL
LIN {X 0,Y 277.82,Z 320.867,A -85,B 0,C 180,E1 -17461.449,E2 -17461.449} C_VEL
LIN {X 0,Y 277.605,Z 320.901,A -85,B 0,C 180,E1 -17467.272,E2 -17467.272} C_VEL
LIN {X 0,Y 277.462,Z 320.923,A -85,B 0,C 180,E1 -17470.213,E2 -17470.213} C_VEL
LIN {X 0,Y 277.413,Z 320.917,A -85,B 0,C 180,E1 -17474.675,E2 -17474.675} C_VEL
LIN {X 0,Y 277.308,Z 320.94,A -85,B 0,C 180,E1 -17479.236,E2 -17479.236} C_VEL
LIN {X 0,Y 277.29,Z 320.939,A -85,B 0,C 180,E1 -17483.924,E2 -17483.924} C_VEL
LIN {X 0,Y 277.267,Z 320.934,A -85,B 0,C 180,E1 -17487.48,E2 -17487.48} C_VEL
LIN {X 0,Y 277.251,Z 320.941,A -85,B 0,C 180,E1 -17490.472,E2 -17490.472} C_VEL
LIN {X 0,Y 277.249,Z 320.946,A -85,B 0,C 180,E1 -17493.895,E2 -17493.895} C_VEL
LIN {X 0,Y 277.268,Z 320.938,A -85,B 0,C 180,E1 -17497.469,E2 -17497.469} C_VEL
LIN {X 0,Y 277.212,Z 320.949,A -85,B 0,C 180,E1 -17501.236,E2 -17501.236} C_VEL
LIN {X 0,Y 277.204,Z 320.951,A -85,B 0,C 180,E1 -17505.226,E2 -17505.226} C_VEL
LIN {X 0,Y 277.224,Z 320.948,A -85,B 0,C 180,E1 -17509.511,E2 -17509.511} C_VEL
LIN {X 0,Y 277.257,Z 320.947,A -85,B 0,C 180,E1 -17512.528,E2 -17512.528} C_VEL
LIN {X 0,Y 277.247,Z 320.945,A -85,B 0,C 180,E1 -17516.103,E2 -17516.103} C_VEL
LIN {X 0,Y 277.263,Z 320.945,A -85,B 0,C 180,E1 -17519.538,E2 -17519.538} C_VEL
LIN {X 0,Y 277.308,Z 320.942,A -85,B 0,C 180,E1 -17522.857,E2 -17522.857} C_VEL
LIN {X 0,Y 277.29,Z 320.943,A -85,B 0,C 180,E1 -17526.075,E2 -17526.075} C_VEL
LIN {X 0,Y 277.336,Z 320.941,A -85,B 0,C 180,E1 -17530.764,E2 -17530.764} C_VEL
LIN {X 0,Y 277.411,Z 320.929,A -85,B 0,C 180,E1 -17535.323,E2 -17535.323} C_VEL
LIN {X 0,Y 277.431,Z 320.957,A -85,B 0,C 180,E1 -17535.886,E2 -17535.886} C_VEL
LIN {X 0,Y 278.279,Z 325.158,A -85,B 0,C 180,E1 -17537.368,E2 -17537.368} C_VEL
LIN {X 0,Y 285.665,Z 345.862,A -85,B 0,C 180,E1 -17538.529,E2 -17538.529} C_VEL
LIN {X 0,Y 288.075,Z 358.817,A -85,B 0,C 180,E1 -17539.055,E2 -17539.055} C_VEL
LIN {X 0,Y 286.137,Z 432.708,A -85,B 0,C 180,E1 -17540.901,E2 -17540.901} C_VEL
LIN {X 0,Y 285.391,Z 445.849,A -85,B 0,C 180,E1 -17541.502,E2 -17541.502} C_VEL
LIN {X 0,Y 284.464,Z 458.483,A -85,B 0,C 180,E1 -17542.368,E2 -17542.368} C_VEL
LIN {X 0,Y 283.415,Z 469.736,A -85,B 0,C 180,E1 -17543.413,E2 -17543.413} C_VEL
LIN {X 0,Y 282.027,Z 481.379,A -85,B 0,C 180,E1 -17544.815,E2 -17544.815} C_VEL
LIN {X 0,Y 280.642,Z 491.859,A -85,B 0,C 180,E1 -17546.409,E2 -17546.409} C_VEL
LIN {X 0,Y 279.248,Z 501.303,A -85,B 0,C 180,E1 -17548.196,E2 -17548.196} C_VEL
LIN {X 0,Y 277.898,Z 510.396,A -85,B 0,C 180,E1 -17550.361,E2 -17550.361} C_VEL
LIN {X 0,Y 276.918,Z 517.718,A -85,B 0,C 180,E1 -17552.544,E2 -17552.544} C_VEL
LIN {X 0,Y 276.235,Z 522.681,A -85,B 0,C 180,E1 -17554.376,E2 -17554.376} C_VEL
LIN {X 0,Y 275.841,Z 527.242,A -85,B 0,C 180,E1 -17556.459,E2 -17556.459} C_VEL
LIN {X 0,Y 275.397,Z 531.188,A -85,B 0,C 180,E1 -17558.806,E2 -17558.806} C_VEL
LIN {X 0,Y 275.192,Z 533.103,A -85,B 0,C 180,E1 -17560.297,E2 -17560.297} C_VEL
LIN {X 0,Y 275.099,Z 534.537,A -85,B 0,C 180,E1 -17561.792,E2 -17561.792} C_VEL
LIN {X 0,Y 275.058,Z 535.857,A -85,B 0,C 180,E1 -17563.848,E2 -17563.848} C_VEL
LIN {X 0,Y 275.128,Z 536.384,A -85,B 0,C 180,E1 -17566.318,E2 -17566.318} C_VEL
LIN {X 0,Y 275.311,Z 536.138,A -85,B 0,C 180,E1 -17567.837,E2 -17567.837} C_VEL
LIN {X 0,Y 275.579,Z 535.487,A -85,B 0,C 180,E1 -17569.36,E2 -17569.36} C_VEL
LIN {X 0,Y 275.909,Z 534.423,A -85,B 0,C 180,E1 -17570.891,E2 -17570.891} C_VEL
LIN {X 0,Y 276.691,Z 531.949,A -85,B 0,C 180,E1 -17573.183,E2 -17573.183} C_VEL
LIN {X 0,Y 277.681,Z 528.391,A -85,B 0,C 180,E1 -17575.483,E2 -17575.483} C_VEL
LIN {X 0,Y 279.026,Z 523.862,A -85,B 0,C 180,E1 -17577.668,E2 -17577.668} C_VEL
LIN {X 0,Y 280.799,Z 517.49,A -85,B 0,C 180,E1 -17580.036,E2 -17580.036} C_VEL
LIN {X 0,Y 282.659,Z 510.912,A -85,B 0,C 180,E1 -17581.972,E2 -17581.972} C_VEL
LIN {X 0,Y 284.929,Z 501.789,A -85,B 0,C 180,E1 -17584.133,E2 -17584.133} C_VEL
LIN {X 0,Y 287.312,Z 491.964,A -85,B 0,C 180,E1 -17585.947,E2 -17585.947} C_VEL
LIN {X 0,Y 289.679,Z 480.93,A -85,B 0,C 180,E1 -17587.556,E2 -17587.556} C_VEL
LIN {X 0,Y 291.602,Z 470.161,A -85,B 0,C 180,E1 -17588.8,E2 -17588.8} C_VEL
LIN {X 0,Y 293.308,Z 458.684,A -85,B 0,C 180,E1 -17589.82,E2 -17589.82} C_VEL
LIN {X 0,Y 294.79,Z 445.379,A -85,B 0,C 180,E1 -17590.683,E2 -17590.683} C_VEL
LIN {X 0,Y 295.672,Z 433.314,A -85,B 0,C 180,E1 -17591.211,E2 -17591.211} C_VEL
LIN {X 0,Y 298.26,Z 365.176,A -85,B 0,C 180,E1 -17592.879,E2 -17592.879} C_VEL
LIN {X 0,Y 291.874,Z 350.73,A -85,B 0,C 180,E1 -17594.156,E2 -17594.156} C_VEL
LIN {X 0,Y 284.292,Z 336.163,A -85,B 0,C 180,E1 -17595.701,E2 -17595.701} C_VEL
LIN {X 0,Y 278.538,Z 325.832,A -85,B 0,C 180,E1 -17596.935,E2 -17596.935} C_VEL
LIN {X 0,Y 277.18,Z 320.961,A -85,B 0,C 180,E1 -17599.087,E2 -17599.087} C_VEL
LIN {X 0,Y 277.253,Z 320.948,A -85,B 0,C 180,E1 -17602.529,E2 -17602.529} C_VEL
LIN {X 0,Y 277.239,Z 320.925,A -85,B 0,C 180,E1 -17606.103,E2 -17606.103} C_VEL
LIN {X 0,Y 277.254,Z 320.948,A -85,B 0,C 180,E1 -17609.538,E2 -17609.538} C_VEL
LIN {X 0,Y 277.281,Z 320.946,A -85,B 0,C 180,E1 -17612.856,E2 -17612.856} C_VEL
LIN {X 0,Y 277.264,Z 320.948,A -85,B 0,C 180,E1 -17616.074,E2 -17616.074} C_VEL
LIN {X 0,Y 277.245,Z 320.946,A -85,B 0,C 180,E1 -17619.086,E2 -17619.086} C_VEL
LIN {X 0,Y 276.646,Z 321.03,A -85,B 0,C 180,E1 -17620.299,E2 -17620.299} C_VEL
LIN {X 0,Y 273.855,Z 321.383,A -85,B 0,C 180,E1 -17622.276,E2 -17622.276} C_VEL
LIN {X 0,Y 271.44,Z 321.676,A -85,B 0,C 180,E1 -17623.883,E2 -17623.883} C_VEL
LIN {X 0,Y 270.388,Z 321.802,A -85,B 0,C 180,E1 -17625.128,E2 -17625.128} C_VEL
LIN {X 0,Y 270.295,Z 321.806,A -85,B 0,C 180,E1 -17625.549,E2 -17625.549} C_VEL
LIN {X 0,Y 270.376,Z 321.804,A -85,B 0,C 180,E1 -17629.517,E2 -17629.517} C_VEL
LIN {X 0,Y 270.552,Z 321.772,A -85,B 0,C 180,E1 -17632.538,E2 -17632.538} C_VEL
LIN {X 0,Y 270.753,Z 321.754,A -85,B 0,C 180,E1 -17638.513,E2 -17638.513} C_VEL
LIN {X 0,Y 270.765,Z 321.744,A -85,B 0,C 180,E1 -17641.488,E2 -17641.488} C_VEL
LIN {X 0,Y 270.557,Z 321.765,A -85,B 0,C 180,E1 -17647.463,E2 -17647.463} C_VEL
LIN {X 0,Y 270.402,Z 321.8,A -85,B 0,C 180,E1 -17650.483,E2 -17650.483} C_VEL
LIN {X 0,Y 270.37,Z 321.8,A -85,B 0,C 180,E1 -17655.067,E2 -17655.067} C_VEL
LIN {X 0,Y 270.272,Z 321.812,A -85,B 0,C 180,E1 -17659.758,E2 -17659.758} C_VEL
LIN {X 0,Y 270.191,Z 321.824,A -85,B 0,C 180,E1 -17664.594,E2 -17664.594} C_VEL
LIN {X 0,Y 270.19,Z 321.818,A -85,B 0,C 180,E1 -17667.918,E2 -17667.918} C_VEL
LIN {X 0,Y 270.167,Z 321.823,A -85,B 0,C 180,E1 -17671.351,E2 -17671.351} C_VEL
LIN {X 0,Y 270.192,Z 321.823,A -85,B 0,C 180,E1 -17674.907,E2 -17674.907} C_VEL
LIN {X 0,Y 270.162,Z 321.826,A -85,B 0,C 180,E1 -17678.704,E2 -17678.704} C_VEL
LIN {X 0,Y 270.143,Z 321.81,A -85,B 0,C 180,E1 -17683.246,E2 -17683.246} C_VEL
LIN {X 0,Y 270.168,Z 321.833,A -85,B 0,C 180,E1 -17687.443,E2 -17687.443} C_VEL
LIN {X 0,Y 270.182,Z 321.869,A -85,B 0,C 180,E1 -17689.557,E2 -17689.557} C_VEL
LIN {X 0,Y 272.448,Z 329.798,A -85,B 0,C 180,E1 -17693.099,E2 -17693.099} C_VEL
LIN {X 0,Y 274.447,Z 337.96,A -85,B 0,C 180,E1 -17696.444,E2 -17696.444} C_VEL
LIN {X 0,Y 276.658,Z 342.266,A -85,B 0,C 180,E1 -17696.962,E2 -17696.962} C_VEL
LIN {X 0,Y 283.809,Z 356.679,A -85,B 0,C 180,E1 -17698.533,E2 -17698.533} C_VEL
LIN {X 0,Y 287.65,Z 365.566,A -85,B 0,C 180,E1 -17699.362,E2 -17699.362} C_VEL
LIN {X 0,Y 291.43,Z 386.622,A -85,B 0,C 180,E1 -17700.512,E2 -17700.512} C_VEL
LIN {X 0,Y 291.512,Z 390.984,A -85,B 0,C 180,E1 -17700.652,E2 -17700.652} C_VEL
LIN {X 0,Y 289.332,Z 447.49,A -85,B 0,C 180,E1 -17702.078,E2 -17702.078} C_VEL
LIN {X 0,Y 288.154,Z 461.07,A -85,B 0,C 180,E1 -17702.69,E2 -17702.69} C_VEL
LIN {X 0,Y 286.418,Z 473.435,A -85,B 0,C 180,E1 -17703.497,E2 -17703.497} C_VEL
LIN {X 0,Y 284.415,Z 485.265,A -85,B 0,C 180,E1 -17704.576,E2 -17704.576} C_VEL
LIN {X 0,Y 282.097,Z 496.638,A -85,B 0,C 180,E1 -17705.925,E2 -17705.925} C_VEL
LIN {X 0,Y 279.699,Z 506.915,A -85,B 0,C 180,E1 -17707.47,E2 -17707.47} C_VEL
LIN {X 0,Y 277.287,Z 516.179,A -85,B 0,C 180,E1 -17709.218,E2 -17709.218} C_VEL
LIN {X 0,Y 275.189,Z 524.103,A -85,B 0,C 180,E1 -17711.081,E2 -17711.081} C_VEL
LIN {X 0,Y 272.946,Z 532.429,A -85,B 0,C 180,E1 -17713.548,E2 -17713.548} C_VEL
LIN {X 0,Y 271.191,Z 538.278,A -85,B 0,C 180,E1 -17715.749,E2 -17715.749} C_VEL
LIN {X 0,Y 269.954,Z 542.907,A -85,B 0,C 180,E1 -17717.98,E2 -17717.98} C_VEL
LIN {X 0,Y 269.058,Z 546.454,A -85,B 0,C 180,E1 -17720.226,E2 -17720.226} C_VEL
LIN {X 0,Y 268.486,Z 549.017,A -85,B 0,C 180,E1 -17722.481,E2 -17722.481} C_VEL
LIN {X 0,Y 268.196,Z 550.659,A -85,B 0,C 180,E1 -17724.738,E2 -17724.738} C_VEL
LIN {X 0,Y 268.158,Z 551.415,A -85,B 0,C 180,E1 -17726.997,E2 -17726.997} C_VEL
LIN {X 0,Y 268.182,Z 551.426,A -85,B 0,C 180,E1 -17728.5,E2 -17728.5} C_VEL
LIN {X 0,Y 268.202,Z 551.051,A -85,B 0,C 180,E1 -17730.001,E2 -17730.001} C_VEL
LIN {X 0,Y 268.196,Z 550.252,A -85,B 0,C 180,E1 -17731.503,E2 -17731.503} C_VEL
LIN {X 0,Y 268.192,Z 549.025,A -85,B 0,C 180,E1 -17733.006,E2 -17733.006} C_VEL
LIN {X 0,Y 268.214,Z 546.346,A -85,B 0,C 180,E1 -17735.302,E2 -17735.302} C_VEL
LIN {X 0,Y 268.424,Z 542.743,A -85,B 0,C 180,E1 -17737.524,E2 -17737.524} C_VEL
LIN {X 0,Y 268.841,Z 537.946,A -85,B 0,C 180,E1 -17739.785,E2 -17739.785} C_VEL
LIN {X 0,Y 269.496,Z 531.861,A -85,B 0,C 180,E1 -17742.043,E2 -17742.043} C_VEL
LIN {X 0,Y 270.637,Z 524.285,A -85,B 0,C 180,E1 -17744.284,E2 -17744.284} C_VEL
LIN {X 0,Y 271.831,Z 516.535,A -85,B 0,C 180,E1 -17746.138,E2 -17746.138} C_VEL
LIN {X 0,Y 273.053,Z 507.048,A -85,B 0,C 180,E1 -17747.992,E2 -17747.992} C_VEL
LIN {X 0,Y 274.517,Z 496.501,A -85,B 0,C 180,E1 -17749.636,E2 -17749.636} C_VEL
LIN {X 0,Y 276.04,Z 484.774,A -85,B 0,C 180,E1 -17751.078,E2 -17751.078} C_VEL
LIN {X 0,Y 277.437,Z 472.276,A -85,B 0,C 180,E1 -17752.236,E2 -17752.236} C_VEL
LIN {X 0,Y 278.551,Z 459.076,A -85,B 0,C 180,E1 -17753.121,E2 -17753.121} C_VEL
LIN {X 0,Y 279.311,Z 445.912,A -85,B 0,C 180,E1 -17753.692,E2 -17753.692} C_VEL
LIN {X 0,Y 280.828,Z 383.116,A -85,B 0,C 180,E1 -17755.3,E2 -17755.3} C_VEL
LIN {X 0,Y 275.624,Z 345.137,A -85,B 0,C 180,E1 -17756.756,E2 -17756.756} C_VEL
LIN {X 0,Y 273.715,Z 339.058,A -85,B 0,C 180,E1 -17757.096,E2 -17757.096} C_VEL
LIN {X 0,Y 271.621,Z 328.231,A -85,B 0,C 180,E1 -17760.733,E2 -17760.733} C_VEL
LIN {X 0,Y 270.237,Z 321.818,A -85,B 0,C 180,E1 -17762.993,E2 -17762.993} C_VEL
LIN {X 0,Y 270.203,Z 321.827,A -85,B 0,C 180,E1 -17766.745,E2 -17766.745} C_VEL
LIN {X 0,Y 270.139,Z 321.835,A -85,B 0,C 180,E1 -17771.02,E2 -17771.02} C_VEL
LIN {X 0,Y 270.151,Z 321.837,A -85,B 0,C 180,E1 -17774.622,E2 -17774.622} C_VEL
LIN {X 0,Y 270.177,Z 321.83,A -85,B 0,C 180,E1 -17777.442,E2 -17777.442} C_VEL
LIN {X 0,Y 270.212,Z 321.823,A -85,B 0,C 180,E1 -17781.375,E2 -17781.375} C_VEL
LIN {X 0,Y 270.206,Z 321.826,A -85,B 0,C 180,E1 -17785.095,E2 -17785.095} C_VEL
LIN {X 0,Y 270.189,Z 321.829,A -85,B 0,C 180,E1 -17789.137,E2 -17789.137} C_VEL
LIN {X 0,Y 270.231,Z 321.82,A -85,B 0,C 180,E1 -17792.162,E2 -17792.162} C_VEL
LIN {X 0,Y 270.235,Z 321.822,A -85,B 0,C 180,E1 -17795.541,E2 -17795.541} C_VEL
LIN {X 0,Y 270.256,Z 321.808,A -85,B 0,C 180,E1 -17800.241,E2 -17800.241} C_VEL
LIN {X 0,Y 270.373,Z 321.804,A -85,B 0,C 180,E1 -17804.933,E2 -17804.933} C_VEL
LIN {X 0,Y 270.417,Z 321.791,A -85,B 0,C 180,E1 -17809.518,E2 -17809.518} C_VEL
LIN {X 0,Y 270.58,Z 321.772,A -85,B 0,C 180,E1 -17812.538,E2 -17812.538} C_VEL
LIN {X 0,Y 270.783,Z 321.75,A -85,B 0,C 180,E1 -17818.512,E2 -17818.512} C_VEL
LIN {X 0,Y 270.785,Z 321.743,A -85,B 0,C 180,E1 -17821.487,E2 -17821.487} C_VEL
LIN {X 0,Y 270.567,Z 321.778,A -85,B 0,C 180,E1 -17827.462,E2 -17827.462} C_VEL
LIN {X 0,Y 270.414,Z 321.801,A -85,B 0,C 180,E1 -17830.482,E2 -17830.482} C_VEL
LIN {X 0,Y 270.372,Z 321.791,A -85,B 0,C 180,E1 -17835.066,E2 -17835.066} C_VEL
LIN {X 0,Y 270.255,Z 321.817,A -85,B 0,C 180,E1 -17839.759,E2 -17839.759} C_VEL
LIN {X 0,Y 270.231,Z 321.82,A -85,B 0,C 180,E1 -17844.589,E2 -17844.589} C_VEL
LIN {X 0,Y 270.2,Z 321.812,A -85,B 0,C 180,E1 -17847.916,E2 -17847.916} C_VEL
LIN {X 0,Y 270.177,Z 321.828,A -85,B 0,C 180,E1 -17851.349,E2 -17851.349} C_VEL
LIN {X 0,Y 270.205,Z 321.823,A -85,B 0,C 180,E1 -17854.905,E2 -17854.905} C_VEL
LIN {X 0,Y 270.2,Z 321.812,A -85,B 0,C 180,E1 -17858.709,E2 -17858.709} C_VEL
LIN {X 0,Y 270.168,Z 321.829,A -85,B 0,C 180,E1 -17863.248,E2 -17863.248} C_VEL
LIN {X 0,Y 270.174,Z 321.822,A -85,B 0,C 180,E1 -17867.441,E2 -17867.441} C_VEL
LIN {X 0,Y 270.209,Z 321.824,A -85,B 0,C 180,E1 -17871.373,E2 -17871.373} C_VEL
LIN {X 0,Y 270.2,Z 321.819,A -85,B 0,C 180,E1 -17875.093,E2 -17875.093} C_VEL
LIN {X 0,Y 270.186,Z 321.826,A -85,B 0,C 180,E1 -17879.135,E2 -17879.135} C_VEL
LIN {X 0,Y 270.228,Z 321.824,A -85,B 0,C 180,E1 -17882.16,E2 -17882.16} C_VEL
LIN {X 0,Y 270.233,Z 321.821,A -85,B 0,C 180,E1 -17885.539,E2 -17885.539} C_VEL
LIN {X 0,Y 270.298,Z 321.816,A -85,B 0,C 180,E1 -17890.243,E2 -17890.243} C_VEL
LIN {X 0,Y 270.391,Z 321.803,A -85,B 0,C 180,E1 -17895.319,E2 -17895.319} C_VEL
LIN {X 0,Y 270.392,Z 321.937,A -85,B 0,C 180,E1 -17895.511,E2 -17895.511} C_VEL
LIN {X 0,Y 271.11,Z 325.346,A -85,B 0,C 180,E1 -17896.754,E2 -17896.754} C_VEL
LIN {X 0,Y 279.25,Z 347.944,A -85,B 0,C 180,E1 -17898.08,E2 -17898.08} C_VEL
LIN {X 0,Y 281.448,Z 359.605,A -85,B 0,C 180,E1 -17898.572,E2 -17898.572} C_VEL
LIN {X 0,Y 279.417,Z 433.151,A -85,B 0,C 180,E1 -17900.452,E2 -17900.452} C_VEL
LIN {X 0,Y 278.626,Z 446.224,A -85,B 0,C 180,E1 -17901.065,E2 -17901.065} C_VEL
LIN {X 0,Y 277.728,Z 458.241,A -85,B 0,C 180,E1 -17901.907,E2 -17901.907} C_VEL
LIN {X 0,Y 276.561,Z 470.334,A -85,B 0,C 180,E1 -17903.056,E2 -17903.056} C_VEL
LIN {X 0,Y 275.112,Z 481.982,A -85,B 0,C 180,E1 -17904.501,E2 -17904.501} C_VEL
LIN {X 0,Y 273.696,Z 492.389,A -85,B 0,C 180,E1 -17906.134,E2 -17906.134} C_VEL
LIN {X 0,Y 272.383,Z 500.913,A -85,B 0,C 180,E1 -17907.781,E2 -17907.781} C_VEL
LIN {X 0,Y 270.994,Z 510.125,A -85,B 0,C 180,E1 -17909.999,E2 -17909.999} C_VEL
LIN {X 0,Y 269.935,Z 517.533,A -85,B 0,C 180,E1 -17912.237,E2 -17912.237} C_VEL
LIN {X 0,Y 269.13,Z 523.479,A -85,B 0,C 180,E1 -17914.492,E2 -17914.492} C_VEL
LIN {X 0,Y 268.747,Z 527.513,A -85,B 0,C 180,E1 -17916.418,E2 -17916.418} C_VEL
LIN {X 0,Y 268.277,Z 531.746,A -85,B 0,C 180,E1 -17919.042,E2 -17919.042} C_VEL
LIN {X 0,Y 268.062,Z 533.561,A -85,B 0,C 180,E1 -17920.574,E2 -17920.574} C_VEL
LIN {X 0,Y 267.992,Z 534.929,A -85,B 0,C 180,E1 -17922.109,E2 -17922.109} C_VEL
LIN {X 0,Y 267.968,Z 536.062,A -85,B 0,C 180,E1 -17923.976,E2 -17923.976} C_VEL
LIN {X 0,Y 268.065,Z 536.561,A -85,B 0,C 180,E1 -17926.76,E2 -17926.76} C_VEL
LIN {X 0,Y 268.53,Z 535.714,A -85,B 0,C 180,E1 -17929.577,E2 -17929.577} C_VEL
LIN {X 0,Y 268.972,Z 534.389,A -85,B 0,C 180,E1 -17931.456,E2 -17931.456} C_VEL
LIN {X 0,Y 270.054,Z 531.01,A -85,B 0,C 180,E1 -17934.377,E2 -17934.377} C_VEL
LIN {X 0,Y 271.43,Z 526.638,A -85,B 0,C 180,E1 -17936.942,E2 -17936.942} C_VEL
LIN {X 0,Y 273.039,Z 521.298,A -85,B 0,C 180,E1 -17939.277,E2 -17939.277} C_VEL
LIN {X 0,Y 275.08,Z 514.484,A -85,B 0,C 180,E1 -17941.582,E2 -17941.582} C_VEL
LIN {X 0,Y 277.423,Z 505.922,A -85,B 0,C 180,E1 -17943.869,E2 -17943.869} C_VEL
LIN {X 0,Y 279.783,Z 497.045,A -85,B 0,C 180,E1 -17945.732,E2 -17945.732} C_VEL
LIN {X 0,Y 282.281,Z 486.446,A -85,B 0,C 180,E1 -17947.496,E2 -17947.496} C_VEL
LIN {X 0,Y 284.623,Z 474.805,A -85,B 0,C 180,E1 -17949.023,E2 -17949.023} C_VEL
LIN {X 0,Y 286.499,Z 463.841,A -85,B 0,C 180,E1 -17950.125,E2 -17950.125} C_VEL
LIN {X 0,Y 288.172,Z 451.349,A -85,B 0,C 180,E1 -17951.073,E2 -17951.073} C_VEL
LIN {X 0,Y 289.275,Z 439.029,A -85,B 0,C 180,E1 -17951.745,E2 -17951.745} C_VEL
LIN {X 0,Y 290.086,Z 425.377,A -85,B 0,C 180,E1 -17952.185,E2 -17952.185} C_VEL
LIN {X 0,Y 292.352,Z 367.281,A -85,B 0,C 180,E1 -17953.599,E2 -17953.599} C_VEL
LIN {X 0,Y 286.141,Z 353.314,A -85,B 0,C 180,E1 -17954.892,E2 -17954.892} C_VEL
LIN {X 0,Y 278.426,Z 338.433,A -85,B 0,C 180,E1 -17956.541,E2 -17956.541} C_VEL
LIN {X 0,Y 272.891,Z 329.067,A -85,B 0,C 180,E1 -17957.763,E2 -17957.763} C_VEL
LIN {X 0,Y 271.271,Z 326.021,A -85,B 0,C 180,E1 -17958.175,E2 -17958.175} C_VEL
LIN {X 0,Y 270.164,Z 321.831,A -85,B 0,C 180,E1 -17960.165,E2 -17960.165} C_VEL
LIN {X 0,Y 270.216,Z 321.829,A -85,B 0,C 180,E1 -17963.73,E2 -17963.73} C_VEL
LIN {X 0,Y 270.194,Z 321.805,A -85,B 0,C 180,E1 -17966.892,E2 -17966.892} C_VEL
LIN {X 0,Y 270.175,Z 321.824,A -85,B 0,C 180,E1 -17970.381,E2 -17970.381} C_VEL
LIN {X 0,Y 270.189,Z 321.822,A -85,B 0,C 180,E1 -17973.756,E2 -17973.756} C_VEL
LIN {X 0,Y 270.184,Z 321.825,A -85,B 0,C 180,E1 -17977.035,E2 -17977.035} C_VEL
LIN {X 0,Y 270.212,Z 321.825,A -85,B 0,C 180,E1 -17980.238,E2 -17980.238} C_VEL
LIN {X 0,Y 270.329,Z 321.809,A -85,B 0,C 180,E1 -17984.932,E2 -17984.932} C_VEL
LIN {X 0,Y 270.295,Z 321.806,A -85,B 0,C 180,E1 -17985.549,E2 -17985.549} C_VEL
LIN {X 0,Y 269.617,Z 321.888,A -85,B 0,C 180,E1 -17986.793,E2 -17986.793} C_VEL
LIN {X 0,Y 266.812,Z 322.248,A -85,B 0,C 180,E1 -17988.823,E2 -17988.823} C_VEL
LIN {X 0,Y 264.487,Z 322.528,A -85,B 0,C 180,E1 -17990.473,E2 -17990.473} C_VEL
LIN {X 0,Y 263.548,Z 322.64,A -85,B 0,C 180,E1 -17991.75,E2 -17991.75} C_VEL
LIN {X 0,Y 263.502,Z 322.647,A -85,B 0,C 180,E1 -17992.181,E2 -17992.181} C_VEL
LIN {X 0,Y 263.473,Z 322.649,A -85,B 0,C 180,E1 -17996.942,E2 -17996.942} C_VEL
LIN {X 0,Y 263.716,Z 322.63,A -85,B 0,C 180,E1 -17998.473,E2 -17998.473} C_VEL
LIN {X 0,Y 263.727,Z 322.62,A -85,B 0,C 180,E1 -18001.527,E2 -18001.527} C_VEL
LIN {X 0,Y 263.521,Z 322.64,A -85,B 0,C 180,E1 -18007.663,E2 -18007.663} C_VEL
LIN {X 0,Y 263.342,Z 322.68,A -85,B 0,C 180,E1 -18010.767,E2 -18010.767} C_VEL
LIN {X 0,Y 263.316,Z 322.682,A -85,B 0,C 180,E1 -18015.48,E2 -18015.48} C_VEL
LIN {X 0,Y 263.236,Z 322.69,A -85,B 0,C 180,E1 -18020.309,E2 -18020.309} C_VEL
LIN {X 0,Y 263.129,Z 322.709,A -85,B 0,C 180,E1 -18025.3,E2 -18025.3} C_VEL
LIN {X 0,Y 263.126,Z 322.703,A -85,B 0,C 180,E1 -18028.736,E2 -18028.736} C_VEL
LIN {X 0,Y 263.122,Z 322.701,A -85,B 0,C 180,E1 -18032.29,E2 -18032.29} C_VEL
LIN {X 0,Y 263.148,Z 322.699,A -85,B 0,C 180,E1 -18035.985,E2 -18035.985} C_VEL
LIN {X 0,Y 263.067,Z 322.714,A -85,B 0,C 180,E1 -18039.88,E2 -18039.88} C_VEL
LIN {X 0,Y 263.077,Z 322.691,A -85,B 0,C 180,E1 -18043.994,E2 -18043.994} C_VEL
LIN {X 0,Y 263.12,Z 322.713,A -85,B 0,C 180,E1 -18048.108,E2 -18048.108} C_VEL
LIN {X 0,Y 263.145,Z 322.945,A -85,B 0,C 180,E1 -18048.539,E2 -18048.539} C_VEL
LIN {X 0,Y 265.649,Z 331.497,A -85,B 0,C 180,E1 -18052.531,E2 -18052.531} C_VEL
LIN {X 0,Y 267.228,Z 337.716,A -85,B 0,C 180,E1 -18055.202,E2 -18055.202} C_VEL
LIN {X 0,Y 269.673,Z 342.363,A -85,B 0,C 180,E1 -18055.798,E2 -18055.798} C_VEL
LIN {X 0,Y 277.364,Z 357.536,A -85,B 0,C 180,E1 -18057.572,E2 -18057.572} C_VEL
LIN {X 0,Y 282.12,Z 368.309,A -85,B 0,C 180,E1 -18058.645,E2 -18058.645} C_VEL
LIN {X 0,Y 285.634,Z 388.15,A -85,B 0,C 180,E1 -18059.763,E2 -18059.763} C_VEL
LIN {X 0,Y 283.923,Z 435.663,A -85,B 0,C 180,E1 -18060.97,E2 -18060.97} C_VEL
LIN {X 0,Y 283.163,Z 451.196,A -85,B 0,C 180,E1 -18061.451,E2 -18061.451} C_VEL
LIN {X 0,Y 281.69,Z 464.233,A -85,B 0,C 180,E1 -18062.11,E2 -18062.11} C_VEL
LIN {X 0,Y 279.965,Z 475.619,A -85,B 0,C 180,E1 -18062.937,E2 -18062.937} C_VEL
LIN {X 0,Y 277.751,Z 487.724,A -85,B 0,C 180,E1 -18064.122,E2 -18064.122} C_VEL
LIN {X 0,Y 275.671,Z 497.322,A -85,B 0,C 180,E1 -18065.327,E2 -18065.327} C_VEL
LIN {X 0,Y 273.181,Z 507.417,A -85,B 0,C 180,E1 -18066.902,E2 -18066.902} C_VEL
LIN {X 0,Y 270.675,Z 516.527,A -85,B 0,C 180,E1 -18068.686,E2 -18068.686} C_VEL
LIN {X 0,Y 268.341,Z 524.839,A -85,B 0,C 180,E1 -18070.722,E2 -18070.722} C_VEL
LIN {X 0,Y 266.133,Z 532.6,A -85,B 0,C 180,E1 -18073.115,E2 -18073.115} C_VEL
LIN {X 0,Y 264.303,Z 538.373,A -85,B 0,C 180,E1 -18075.369,E2 -18075.369} C_VEL
LIN {X 0,Y 262.994,Z 542.938,A -85,B 0,C 180,E1 -18077.657,E2 -18077.657} C_VEL
LIN {X 0,Y 262.316,Z 545.359,A -85,B 0,C 180,E1 -18079.192,E2 -18079.192} C_VEL
LIN {X 0,Y 261.418,Z 548.938,A -85,B 0,C 180,E1 -18082.276,E2 -18082.276} C_VEL
LIN {X 0,Y 261.086,Z 550.67,A -85,B 0,C 180,E1 -18084.864,E2 -18084.864} C_VEL
LIN {X 0,Y 261.054,Z 551.229,A -85,B 0,C 180,E1 -18086.915,E2 -18086.915} C_VEL
LIN {X 0,Y 261.109,Z 551.214,A -85,B 0,C 180,E1 -18088.459,E2 -18088.459} C_VEL
LIN {X 0,Y 261.128,Z 550.807,A -85,B 0,C 180,E1 -18090.001,E2 -18090.001} C_VEL
LIN {X 0,Y 261.123,Z 549.96,A -85,B 0,C 180,E1 -18091.544,E2 -18091.544} C_VEL
LIN {X 0,Y 261.105,Z 548.705,A -85,B 0,C 180,E1 -18093.087,E2 -18093.087} C_VEL
LIN {X 0,Y 261.126,Z 546.267,A -85,B 0,C 180,E1 -18095.232,E2 -18095.232} C_VEL
LIN {X 0,Y 261.354,Z 542.304,A -85,B 0,C 180,E1 -18097.728,E2 -18097.728} C_VEL
LIN {X 0,Y 261.794,Z 537.441,A -85,B 0,C 180,E1 -18100.051,E2 -18100.051} C_VEL
LIN {X 0,Y 262.515,Z 531.285,A -85,B 0,C 180,E1 -18102.368,E2 -18102.368} C_VEL
LIN {X 0,Y 263.722,Z 523.628,A -85,B 0,C 180,E1 -18104.666,E2 -18104.666} C_VEL
LIN {X 0,Y 264.983,Z 515.774,A -85,B 0,C 180,E1 -18106.567,E2 -18106.567} C_VEL
LIN {X 0,Y 266.215,Z 506.12,A -85,B 0,C 180,E1 -18108.471,E2 -18108.471} C_VEL
LIN {X 0,Y 267.599,Z 496.735,A -85,B 0,C 180,E1 -18109.965,E2 -18109.965} C_VEL
LIN {X 0,Y 269.156,Z 485.102,A -85,B 0,C 180,E1 -18111.443,E2 -18111.443} C_VEL
LIN {X 0,Y 270.596,Z 472.829,A -85,B 0,C 180,E1 -18112.627,E2 -18112.627} C_VEL
LIN {X 0,Y 271.824,Z 459.131,A -85,B 0,C 180,E1 -18113.576,E2 -18113.576} C_VEL
LIN {X 0,Y 272.598,Z 446.2,A -85,B 0,C 180,E1 -18114.161,E2 -18114.161} C_VEL
LIN {X 0,Y 274.176,Z 383.932,A -85,B 0,C 180,E1 -18115.794,E2 -18115.794} C_VEL
LIN {X 0,Y 269.25,Z 347.164,A -85,B 0,C 180,E1 -18117.238,E2 -18117.238} C_VEL
LIN {X 0,Y 266.493,Z 338.821,A -85,B 0,C 180,E1 -18117.739,E2 -18117.739} C_VEL
LIN {X 0,Y 264.232,Z 327.535,A -85,B 0,C 180,E1 -18121.664,E2 -18121.664} C_VEL
LIN {X 0,Y 263.182,Z 322.699,A -85,B 0,C 180,E1 -18123.421,E2 -18123.421} C_VEL
LIN {X 0,Y 263.155,Z 322.705,A -85,B 0,C 180,E1 -18126.755,E2 -18126.755} C_VEL
LIN {X 0,Y 263.077,Z 322.717,A -85,B 0,C 180,E1 -18129.879,E2 -18129.879} C_VEL
LIN {X 0,Y 263.103,Z 322.714,A -85,B 0,C 180,E1 -18133.99,E2 -18133.99} C_VEL
LIN {X 0,Y 263.129,Z 322.711,A -85,B 0,C 180,E1 -18138.407,E2 -18138.407} C_VEL
LIN {X 0,Y 263.187,Z 322.701,A -85,B 0,C 180,E1 -18143.237,E2 -18143.237} C_VEL
LIN {X 0,Y 263.133,Z 322.705,A -85,B 0,C 180,E1 -18147.711,E2 -18147.711} C_VEL
LIN {X 0,Y 263.16,Z 322.702,A -85,B 0,C 180,E1 -18151.802,E2 -18151.802} C_VEL
LIN {X 0,Y 263.197,Z 322.702,A -85,B 0,C 180,E1 -18155.217,E2 -18155.217} C_VEL
LIN {X 0,Y 263.24,Z 322.683,A -85,B 0,C 180,E1 -18159.691,E2 -18159.691} C_VEL
LIN {X 0,Y 263.315,Z 322.682,A -85,B 0,C 180,E1 -18164.519,E2 -18164.519} C_VEL
LIN {X 0,Y 263.359,Z 322.672,A -85,B 0,C 180,E1 -18169.233,E2 -18169.233} C_VEL
LIN {X 0,Y 263.542,Z 322.649,A -85,B 0,C 180,E1 -18172.337,E2 -18172.337} C_VEL
LIN {X 0,Y 263.746,Z 322.627,A -85,B 0,C 180,E1 -18178.473,E2 -18178.473} C_VEL
LIN {X 0,Y 263.748,Z 322.619,A -85,B 0,C 180,E1 -18181.527,E2 -18181.527} C_VEL
LIN {X 0,Y 263.531,Z 322.655,A -85,B 0,C 180,E1 -18187.662,E2 -18187.662} C_VEL
LIN {X 0,Y 263.357,Z 322.677,A -85,B 0,C 180,E1 -18190.766,E2 -18190.766} C_VEL
LIN {X 0,Y 263.314,Z 322.667,A -85,B 0,C 180,E1 -18195.48,E2 -18195.48} C_VEL
LIN {X 0,Y 263.239,Z 322.691,A -85,B 0,C 180,E1 -18200.308,E2 -18200.308} C_VEL
LIN {X 0,Y 263.173,Z 322.694,A -85,B 0,C 180,E1 -18205.295,E2 -18205.295} C_VEL
LIN {X 0,Y 263.137,Z 322.691,A -85,B 0,C 180,E1 -18208.734,E2 -18208.734} C_VEL
LIN {X 0,Y 263.131,Z 322.703,A -85,B 0,C 180,E1 -18212.288,E2 -18212.288} C_VEL
LIN {X 0,Y 263.185,Z 322.692,A -85,B 0,C 180,E1 -18216.762,E2 -18216.762} C_VEL
LIN {X 0,Y 263.127,Z 322.705,A -85,B 0,C 180,E1 -18221.592,E2 -18221.592} C_VEL
LIN {X 0,Y 263.125,Z 322.708,A -85,B 0,C 180,E1 -18223.983,E2 -18223.983} C_VEL
LIN {X 0,Y 263.126,Z 322.703,A -85,B 0,C 180,E1 -18228.406,E2 -18228.406} C_VEL
LIN {X 0,Y 263.159,Z 322.706,A -85,B 0,C 180,E1 -18232.102,E2 -18232.102} C_VEL
LIN {X 0,Y 263.153,Z 322.698,A -85,B 0,C 180,E1 -18235.884,E2 -18235.884} C_VEL
LIN {X 0,Y 263.129,Z 322.705,A -85,B 0,C 180,E1 -18239.503,E2 -18239.503} C_VEL
LIN {X 0,Y 263.156,Z 322.704,A -85,B 0,C 180,E1 -18242.997,E2 -18242.997} C_VEL
LIN {X 0,Y 263.154,Z 322.706,A -85,B 0,C 180,E1 -18246.383,E2 -18246.383} C_VEL
LIN {X 0,Y 263.263,Z 322.692,A -85,B 0,C 180,E1 -18249.692,E2 -18249.692} C_VEL
LIN {X 0,Y 263.352,Z 322.783,A -85,B 0,C 180,E1 -18255.065,E2 -18255.065} C_VEL
LIN {X 0,Y 263.953,Z 325.551,A -85,B 0,C 180,E1 -18256.109,E2 -18256.109} C_VEL
LIN {X 0,Y 272.171,Z 348.058,A -85,B 0,C 180,E1 -18257.496,E2 -18257.496} C_VEL
LIN {X 0,Y 273.601,Z 353.488,A -85,B 0,C 180,E1 -18257.77,E2 -18257.77} C_VEL
LIN {X 0,Y 274.824,Z 361.358,A -85,B 0,C 180,E1 -18258.091,E2 -18258.091} C_VEL
LIN {X 0,Y 272.691,Z 433.617,A -85,B 0,C 180,E1 -18259.98,E2 -18259.98} C_VEL
LIN {X 0,Y 271.843,Z 447.346,A -85,B 0,C 180,E1 -18260.653,E2 -18260.653} C_VEL
LIN {X 0,Y 270.812,Z 460.166,A -85,B 0,C 180,E1 -18261.605,E2 -18261.605} C_VEL
LIN {X 0,Y 269.495,Z 472.978,A -85,B 0,C 180,E1 -18262.919,E2 -18262.919} C_VEL
LIN {X 0,Y 268.041,Z 483.867,A -85,B 0,C 180,E1 -18264.356,E2 -18264.356} C_VEL
LIN {X 0,Y 266.772,Z 492.908,A -85,B 0,C 180,E1 -18265.844,E2 -18265.844} C_VEL
LIN {X 0,Y 265.271,Z 502.204,A -85,B 0,C 180,E1 -18267.721,E2 -18267.721} C_VEL
LIN {X 0,Y 263.842,Z 511.215,A -85,B 0,C 180,E1 -18269.999,E2 -18269.999} C_VEL
LIN {X 0,Y 262.8,Z 518.465,A -85,B 0,C 180,E1 -18272.298,E2 -18272.298} C_VEL
LIN {X 0,Y 262.023,Z 524.252,A -85,B 0,C 180,E1 -18274.614,E2 -18274.614} C_VEL
LIN {X 0,Y 261.576,Z 528.673,A -85,B 0,C 180,E1 -18276.865,E2 -18276.865} C_VEL
LIN {X 0,Y 261.141,Z 532.276,A -85,B 0,C 180,E1 -18279.291,E2 -18279.291} C_VEL
LIN {X 0,Y 260.935,Z 534.004,A -85,B 0,C 180,E1 -18280.866,E2 -18280.866} C_VEL
LIN {X 0,Y 260.873,Z 535.319,A -85,B 0,C 180,E1 -18282.445,E2 -18282.445} C_VEL
LIN {X 0,Y 260.878,Z 536.265,A -85,B 0,C 180,E1 -18284.111,E2 -18284.111} C_VEL
LIN {X 0,Y 260.896,Z 536.689,A -85,B 0,C 180,E1 -18285.626,E2 -18285.626} C_VEL
LIN {X 0,Y 261.012,Z 536.738,A -85,B 0,C 180,E1 -18287.227,E2 -18287.227} C_VEL
LIN {X 0,Y 261.477,Z 535.931,A -85,B 0,C 180,E1 -18289.826,E2 -18289.826} C_VEL
LIN {X 0,Y 262.069,Z 534.346,A -85,B 0,C 180,E1 -18292.05,E2 -18292.05} C_VEL
LIN {X 0,Y 263.101,Z 531.27,A -85,B 0,C 180,E1 -18294.741,E2 -18294.741} C_VEL
LIN {X 0,Y 264.272,Z 527.828,A -85,B 0,C 180,E1 -18296.876,E2 -18296.876} C_VEL
LIN {X 0,Y 265.92,Z 522.742,A -85,B 0,C 180,E1 -18299.29,E2 -18299.29} C_VEL
LIN {X 0,Y 267.978,Z 516.366,A -85,B 0,C 180,E1 -18301.634,E2 -18301.634} C_VEL
LIN {X 0,Y 269.925,Z 509.774,A -85,B 0,C 180,E1 -18303.574,E2 -18303.574} C_VEL
LIN {X 0,Y 272.234,Z 501.661,A -85,B 0,C 180,E1 -18305.509,E2 -18305.509} C_VEL
LIN {X 0,Y 274.93,Z 491.332,A -85,B 0,C 180,E1 -18307.454,E2 -18307.454} C_VEL
LIN {X 0,Y 277.4,Z 480.524,A -85,B 0,C 180,E1 -18309.064,E2 -18309.064} C_VEL
LIN {X 0,Y 279.525,Z 469.522,A -85,B 0,C 180,E1 -18310.345,E2 -18310.345} C_VEL
LIN {X 0,Y 281.45,Z 457.354,A -85,B 0,C 180,E1 -18311.422,E2 -18311.422} C_VEL
LIN {X 0,Y 282.925,Z 444.198,A -85,B 0,C 180,E1 -18312.278,E2 -18312.278} C_VEL
LIN {X 0,Y 283.864,Z 431.765,A -85,B 0,C 180,E1 -18312.795,E2 -18312.795} C_VEL
LIN {X 0,Y 286.427,Z 369.187,A -85,B 0,C 180,E1 -18314.365,E2 -18314.365} C_VEL
LIN {X 0,Y 280.59,Z 356.168,A -85,B 0,C 180,E1 -18315.632,E2 -18315.632} C_VEL
LIN {X 0,Y 273.443,Z 342.428,A -85,B 0,C 180,E1 -18317.222,E2 -18317.222} C_VEL
LIN {X 0,Y 266.548,Z 330.552,A -85,B 0,C 180,E1 -18318.827,E2 -18318.827} C_VEL
LIN {X 0,Y 264.217,Z 326.715,A -85,B 0,C 180,E1 -18319.394,E2 -18319.394} C_VEL
LIN {X 0,Y 264.009,Z 326.139,A -85,B 0,C 180,E1 -18319.544,E2 -18319.544} C_VEL
LIN {X 0,Y 263.147,Z 322.71,A -85,B 0,C 180,E1 -18321.27,E2 -18321.27} C_VEL
LIN {X 0,Y 263.154,Z 322.703,A -85,B 0,C 180,E1 -18324.017,E2 -18324.017} C_VEL
LIN {X 0,Y 263.12,Z 322.694,A -85,B 0,C 180,E1 -18327.71,E2 -18327.71} C_VEL
LIN {X 0,Y 263.139,Z 322.706,A -85,B 0,C 180,E1 -18331.805,E2 -18331.805} C_VEL
LIN {X 0,Y 263.179,Z 322.699,A -85,B 0,C 180,E1 -18335.219,E2 -18335.219} C_VEL
LIN {X 0,Y 263.2,Z 322.7,A -85,B 0,C 180,E1 -18339.689,E2 -18339.689} C_VEL
LIN {X 0,Y 263.279,Z 322.688,A -85,B 0,C 180,E1 -18344.518,E2 -18344.518} C_VEL
LIN {X 0,Y 263.321,Z 322.682,A -85,B 0,C 180,E1 -18349.233,E2 -18349.233} C_VEL
LIN {X 0,Y 263.502,Z 322.647,A -85,B 0,C 180,E1 -18352.181,E2 -18352.181} C_VEL
LIN {X 0,Y 262.932,Z 322.73,A -85,B 0,C 180,E1 -18353.455,E2 -18353.455} C_VEL
LIN {X 0,Y 260.175,Z 323.07,A -85,B 0,C 180,E1 -18355.533,E2 -18355.533} C_VEL
LIN {X 0,Y 257.781,Z 323.367,A -85,B 0,C 180,E1 -18357.222,E2 -18357.222} C_VEL
LIN {X 0,Y 256.745,Z 323.498,A -85,B 0,C 180,E1 -18358.531,E2 -18358.531} C_VEL
LIN {X 0,Y 256.658,Z 323.508,A -85,B 0,C 180,E1 -18358.975,E2 -18358.975} C_VEL
LIN {X 0,Y 256.689,Z 323.496,A -85,B 0,C 180,E1 -18361.569,E2 -18361.569} C_VEL
LIN {X 0,Y 256.449,Z 323.532,A -85,B 0,C 180,E1 -18366.294,E2 -18366.294} C_VEL
LIN {X 0,Y 256.42,Z 323.537,A -85,B 0,C 180,E1 -18369.466,E2 -18369.466} C_VEL
LIN {X 0,Y 256.229,Z 323.554,A -85,B 0,C 180,E1 -18374.292,E2 -18374.292} C_VEL
LIN {X 0,Y 256.173,Z 323.558,A -85,B 0,C 180,E1 -18377.565,E2 -18377.565} C_VEL
LIN {X 0,Y 256.133,Z 323.577,A -85,B 0,C 180,E1 -18381.11,E2 -18381.11} C_VEL
LIN {X 0,Y 256.098,Z 323.582,A -85,B 0,C 180,E1 -18385.099,E2 -18385.099} C_VEL
LIN {X 0,Y 256.083,Z 323.579,A -85,B 0,C 180,E1 -18388.576,E2 -18388.576} C_VEL
LIN {X 0,Y 256.068,Z 323.578,A -85,B 0,C 180,E1 -18391.702,E2 -18391.702} C_VEL
LIN {X 0,Y 256.072,Z 323.58,A -85,B 0,C 180,E1 -18395.195,E2 -18395.195} C_VEL
LIN {X 0,Y 256.037,Z 323.585,A -85,B 0,C 180,E1 -18399.149,E2 -18399.149} C_VEL
LIN {X 0,Y 256.019,Z 323.568,A -85,B 0,C 180,E1 -18403.337,E2 -18403.337} C_VEL
LIN {X 0,Y 256.068,Z 323.632,A -85,B 0,C 180,E1 -18407.257,E2 -18407.257} C_VEL
LIN {X 0,Y 258.499,Z 331.829,A -85,B 0,C 180,E1 -18411.297,E2 -18411.297} C_VEL
LIN {X 0,Y 260.07,Z 337.715,A -85,B 0,C 180,E1 -18413.874,E2 -18413.874} C_VEL
LIN {X 0,Y 262.439,Z 342.051,A -85,B 0,C 180,E1 -18414.484,E2 -18414.484} C_VEL
LIN {X 0,Y 270.127,Z 356.73,A -85,B 0,C 180,E1 -18416.363,E2 -18416.363} C_VEL
LIN {X 0,Y 276.529,Z 370.742,A -85,B 0,C 180,E1 -18417.869,E2 -18417.869} C_VEL
LIN {X 0,Y 279.861,Z 389.614,A -85,B 0,C 180,E1 -18418.978,E2 -18418.978} C_VEL
LIN {X 0,Y 277.523,Z 447.079,A -85,B 0,C 180,E1 -18420.488,E2 -18420.488} C_VEL
LIN {X 0,Y 276.249,Z 460.361,A -85,B 0,C 180,E1 -18421.096,E2 -18421.096} C_VEL
LIN {X 0,Y 274.411,Z 472.809,A -85,B 0,C 180,E1 -18421.928,E2 -18421.928} C_VEL
LIN {X 0,Y 272.412,Z 483.912,A -85,B 0,C 180,E1 -18422.955,E2 -18422.955} C_VEL
LIN {X 0,Y 269.798,Z 495.462,A -85,B 0,C 180,E1 -18424.339,E2 -18424.339} C_VEL
LIN {X 0,Y 267.304,Z 505.855,A -85,B 0,C 180,E1 -18425.952,E2 -18425.952} C_VEL
LIN {X 0,Y 264.598,Z 515.263,A -85,B 0,C 180,E1 -18427.761,E2 -18427.761} C_VEL
LIN {X 0,Y 261.934,Z 524.025,A -85,B 0,C 180,E1 -18429.901,E2 -18429.901} C_VEL
LIN {X 0,Y 259.727,Z 531.67,A -85,B 0,C 180,E1 -18432.279,E2 -18432.279} C_VEL
LIN {X 0,Y 257.429,Z 538.455,A -85,B 0,C 180,E1 -18434.97,E2 -18434.97} C_VEL
LIN {X 0,Y 256.026,Z 542.954,A -85,B 0,C 180,E1 -18437.316,E2 -18437.316} C_VEL
LIN {X 0,Y 255.324,Z 545.337,A -85,B 0,C 180,E1 -18438.892,E2 -18438.892} C_VEL
LIN {X 0,Y 254.366,Z 548.859,A -85,B 0,C 180,E1 -18442.061,E2 -18442.061} C_VEL
LIN {X 0,Y 253.975,Z 550.702,A -85,B 0,C 180,E1 -18445.24,E2 -18445.24} C_VEL
LIN {X 0,Y 254.014,Z 551.001,A -85,B 0,C 180,E1 -18448.416,E2 -18448.416} C_VEL
LIN {X 0,Y 254.055,Z 550.549,A -85,B 0,C 180,E1 -18450.001,E2 -18450.001} C_VEL
LIN {X 0,Y 254.052,Z 549.668,A -85,B 0,C 180,E1 -18451.587,E2 -18451.587} C_VEL
LIN {X 0,Y 254.002,Z 548.384,A -85,B 0,C 180,E1 -18453.174,E2 -18453.174} C_VEL
LIN {X 0,Y 254.023,Z 546.237,A -85,B 0,C 180,E1 -18455.12,E2 -18455.12} C_VEL
LIN {X 0,Y 254.31,Z 541.867,A -85,B 0,C 180,E1 -18457.944,E2 -18457.944} C_VEL
LIN {X 0,Y 254.763,Z 536.937,A -85,B 0,C 180,E1 -18460.331,E2 -18460.331} C_VEL
LIN {X 0,Y 255.544,Z 530.71,A -85,B 0,C 180,E1 -18462.711,E2 -18462.711} C_VEL
LIN {X 0,Y 256.801,Z 522.947,A -85,B 0,C 180,E1 -18465.071,E2 -18465.071} C_VEL
LIN {X 0,Y 258.356,Z 513.167,A -85,B 0,C 180,E1 -18467.413,E2 -18467.413} C_VEL
LIN {X 0,Y 259.748,Z 503.021,A -85,B 0,C 180,E1 -18469.358,E2 -18469.358} C_VEL
LIN {X 0,Y 261.465,Z 491.537,A -85,B 0,C 180,E1 -18471.071,E2 -18471.071} C_VEL
LIN {X 0,Y 262.989,Z 480.263,A -85,B 0,C 180,E1 -18472.385,E2 -18472.385} C_VEL
LIN {X 0,Y 264.364,Z 467.589,A -85,B 0,C 180,E1 -18473.503,E2 -18473.503} C_VEL
LIN {X 0,Y 265.465,Z 453.993,A -85,B 0,C 180,E1 -18474.332,E2 -18474.332} C_VEL
LIN {X 0,Y 266.138,Z 440.356,A -85,B 0,C 180,E1 -18474.839,E2 -18474.839} C_VEL
LIN {X 0,Y 267.57,Z 384.833,A -85,B 0,C 180,E1 -18476.308,E2 -18476.308} C_VEL
LIN {X 0,Y 262.858,Z 349.174,A -85,B 0,C 180,E1 -18477.749,E2 -18477.749} C_VEL
LIN {X 0,Y 259.262,Z 338.541,A -85,B 0,C 180,E1 -18478.436,E2 -18478.436} C_VEL
LIN {X 0,Y 256.92,Z 327.194,A -85,B 0,C 180,E1 -18482.525,E2 -18482.525} C_VEL
LIN {X 0,Y 256.131,Z 323.581,A -85,B 0,C 180,E1 -18483.943,E2 -18483.943} C_VEL
LIN {X 0,Y 256.091,Z 323.585,A -85,B 0,C 180,E1 -18487.263,E2 -18487.263} C_VEL
LIN {X 0,Y 256.013,Z 323.594,A -85,B 0,C 180,E1 -18491.213,E2 -18491.213} C_VEL
LIN {X 0,Y 256.045,Z 323.591,A -85,B 0,C 180,E1 -18495.535,E2 -18495.535} C_VEL
LIN {X 0,Y 256.059,Z 323.591,A -85,B 0,C 180,E1 -18498.797,E2 -18498.797} C_VEL
LIN {X 0,Y 256.135,Z 323.582,A -85,B 0,C 180,E1 -18502.868,E2 -18502.868} C_VEL
LIN {X 0,Y 256.071,Z 323.589,A -85,B 0,C 180,E1 -18506.707,E2 -18506.707} C_VEL
LIN {X 0,Y 256.062,Z 323.587,A -85,B 0,C 180,E1 -18510.393,E2 -18510.393} C_VEL
LIN {X 0,Y 256.165,Z 323.576,A -85,B 0,C 180,E1 -18514.876,E2 -18514.876} C_VEL
LIN {X 0,Y 256.153,Z 323.568,A -85,B 0,C 180,E1 -18519.103,E2 -18519.103} C_VEL
LIN {X 0,Y 256.235,Z 323.565,A -85,B 0,C 180,E1 -18524.081,E2 -18524.081} C_VEL
LIN {X 0,Y 256.294,Z 323.559,A -85,B 0,C 180,E1 -18527.327,E2 -18527.327} C_VEL
LIN {X 0,Y 256.503,Z 323.524,A -85,B 0,C 180,E1 -18532.126,E2 -18532.126} C_VEL
LIN {X 0,Y 256.465,Z 323.535,A -85,B 0,C 180,E1 -18536.858,E2 -18536.858} C_VEL
LIN {X 0,Y 256.754,Z 323.495,A -85,B 0,C 180,E1 -18540,E2 -18540} C_VEL
LIN {X 0,Y 256.468,Z 323.52,A -85,B 0,C 180,E1 -18543.141,E2 -18543.141} C_VEL
LIN {X 0,Y 256.495,Z 323.532,A -85,B 0,C 180,E1 -18547.874,E2 -18547.874} C_VEL
LIN {X 0,Y 256.299,Z 323.554,A -85,B 0,C 180,E1 -18551.066,E2 -18551.066} C_VEL
LIN {X 0,Y 256.236,Z 323.553,A -85,B 0,C 180,E1 -18554.291,E2 -18554.291} C_VEL
LIN {X 0,Y 256.172,Z 323.566,A -85,B 0,C 180,E1 -18557.564,E2 -18557.564} C_VEL
LIN {X 0,Y 256.145,Z 323.579,A -85,B 0,C 180,E1 -18561.11,E2 -18561.11} C_VEL
LIN {X 0,Y 256.138,Z 323.571,A -85,B 0,C 180,E1 -18565.112,E2 -18565.112} C_VEL
LIN {X 0,Y 256.059,Z 323.58,A -85,B 0,C 180,E1 -18569.606,E2 -18569.606} C_VEL
LIN {X 0,Y 256.069,Z 323.587,A -85,B 0,C 180,E1 -18573.292,E2 -18573.292} C_VEL
LIN {X 0,Y 256.117,Z 323.571,A -85,B 0,C 180,E1 -18577.27,E2 -18577.27} C_VEL
LIN {X 0,Y 256.057,Z 323.583,A -85,B 0,C 180,E1 -18581.203,E2 -18581.203} C_VEL
LIN {X 0,Y 256.047,Z 323.588,A -85,B 0,C 180,E1 -18585.532,E2 -18585.532} C_VEL
LIN {X 0,Y 256.056,Z 323.582,A -85,B 0,C 180,E1 -18588.795,E2 -18588.795} C_VEL
LIN {X 0,Y 256.128,Z 323.577,A -85,B 0,C 180,E1 -18592.866,E2 -18592.866} C_VEL
LIN {X 0,Y 256.068,Z 323.587,A -85,B 0,C 180,E1 -18596.706,E2 -18596.706} C_VEL
LIN {X 0,Y 256.06,Z 323.591,A -85,B 0,C 180,E1 -18600.392,E2 -18600.392} C_VEL
LIN {X 0,Y 256.164,Z 323.577,A -85,B 0,C 180,E1 -18604.873,E2 -18604.873} C_VEL
LIN {X 0,Y 256.166,Z 323.578,A -85,B 0,C 180,E1 -18609.103,E2 -18609.103} C_VEL
LIN {X 0,Y 256.26,Z 323.564,A -85,B 0,C 180,E1 -18614.081,E2 -18614.081} C_VEL
LIN {X 0,Y 256.299,Z 323.621,A -85,B 0,C 180,E1 -18614.594,E2 -18614.594} C_VEL
LIN {X 0,Y 256.763,Z 325.787,A -85,B 0,C 180,E1 -18615.433,E2 -18615.433} C_VEL
LIN {X 0,Y 265.399,Z 348.961,A -85,B 0,C 180,E1 -18616.935,E2 -18616.935} C_VEL
LIN {X 0,Y 267.181,Z 355.496,A -85,B 0,C 180,E1 -18617.28,E2 -18617.28} C_VEL
LIN {X 0,Y 268.219,Z 361.57,A -85,B 0,C 180,E1 -18617.544,E2 -18617.544} C_VEL
LIN {X 0,Y 266.075,Z 432.904,A -85,B 0,C 180,E1 -18619.44,E2 -18619.44} C_VEL
LIN {X 0,Y 265.32,Z 445.411,A -85,B 0,C 180,E1 -18620.036,E2 -18620.036} C_VEL
LIN {X 0,Y 264.208,Z 458.887,A -85,B 0,C 180,E1 -18621.008,E2 -18621.008} C_VEL
LIN {X 0,Y 263.082,Z 470.179,A -85,B 0,C 180,E1 -18622.13,E2 -18622.13} C_VEL
LIN {X 0,Y 261.561,Z 481.509,A -85,B 0,C 180,E1 -18623.581,E2 -18623.581} C_VEL
LIN {X 0,Y 259.965,Z 492.368,A -85,B 0,C 180,E1 -18625.347,E2 -18625.347} C_VEL
LIN {X 0,Y 258.437,Z 501.83,A -85,B 0,C 180,E1 -18627.271,E2 -18627.271} C_VEL
LIN {X 0,Y 256.948,Z 510.936,A -85,B 0,C 180,E1 -18629.607,E2 -18629.607} C_VEL
LIN {X 0,Y 255.825,Z 518.273,A -85,B 0,C 180,E1 -18631.966,E2 -18631.966} C_VEL
LIN {X 0,Y 255.062,Z 523.245,A -85,B 0,C 180,E1 -18633.949,E2 -18633.949} C_VEL
LIN {X 0,Y 254.58,Z 528.122,A -85,B 0,C 180,E1 -18636.374,E2 -18636.374} C_VEL
LIN {X 0,Y 254.14,Z 531.766,A -85,B 0,C 180,E1 -18638.747,E2 -18638.747} C_VEL
LIN {X 0,Y 253.814,Z 534.448,A -85,B 0,C 180,E1 -18641.175,E2 -18641.175} C_VEL
LIN {X 0,Y 253.76,Z 535.71,A -85,B 0,C 180,E1 -18642.799,E2 -18642.799} C_VEL
LIN {X 0,Y 253.785,Z 536.525,A -85,B 0,C 180,E1 -18644.431,E2 -18644.431} C_VEL
LIN {X 0,Y 253.827,Z 536.92,A -85,B 0,C 180,E1 -18646.073,E2 -18646.073} C_VEL
LIN {X 0,Y 253.972,Z 536.915,A -85,B 0,C 180,E1 -18647.72,E2 -18647.72} C_VEL
LIN {X 0,Y 254.436,Z 536.146,A -85,B 0,C 180,E1 -18650.093,E2 -18650.093} C_VEL
LIN {X 0,Y 255.172,Z 534.304,A -85,B 0,C 180,E1 -18652.679,E2 -18652.679} C_VEL
LIN {X 0,Y 256.167,Z 531.529,A -85,B 0,C 180,E1 -18655.129,E2 -18655.129} C_VEL
LIN {X 0,Y 257.629,Z 527.551,A -85,B 0,C 180,E1 -18657.628,E2 -18657.628} C_VEL
LIN {X 0,Y 259.528,Z 521.98,A -85,B 0,C 180,E1 -18660.252,E2 -18660.252} C_VEL
LIN {X 0,Y 261.619,Z 515.784,A -85,B 0,C 180,E1 -18662.496,E2 -18662.496} C_VEL
LIN {X 0,Y 264.074,Z 507.727,A -85,B 0,C 180,E1 -18664.809,E2 -18664.809} C_VEL
LIN {X 0,Y 266.732,Z 498.816,A -85,B 0,C 180,E1 -18666.827,E2 -18666.827} C_VEL
LIN {X 0,Y 269.281,Z 489.214,A -85,B 0,C 180,E1 -18668.566,E2 -18668.566} C_VEL
LIN {X 0,Y 271.637,Z 478.865,A -85,B 0,C 180,E1 -18670.058,E2 -18670.058} C_VEL
LIN {X 0,Y 273.871,Z 467.35,A -85,B 0,C 180,E1 -18671.358,E2 -18671.358} C_VEL
LIN {X 0,Y 275.728,Z 455.886,A -85,B 0,C 180,E1 -18672.339,E2 -18672.339} C_VEL
LIN {X 0,Y 277.133,Z 442.861,A -85,B 0,C 180,E1 -18673.16,E2 -18673.16} C_VEL
LIN {X 0,Y 278.095,Z 429.85,A -85,B 0,C 180,E1 -18673.669,E2 -18673.669} C_VEL
LIN {X 0,Y 280.587,Z 371.262,A -85,B 0,C 180,E1 -18675.154,E2 -18675.154} C_VEL
LIN {X 0,Y 274.985,Z 358.884,A -85,B 0,C 180,E1 -18676.426,E2 -18676.426} C_VEL
LIN {X 0,Y 268.362,Z 346.062,A -85,B 0,C 180,E1 -18677.967,E2 -18677.967} C_VEL
LIN {X 0,Y 261.918,Z 334.986,A -85,B 0,C 180,E1 -18679.533,E2 -18679.533} C_VEL
LIN {X 0,Y 256.854,Z 326.483,A -85,B 0,C 180,E1 -18680.907,E2 -18680.907} C_VEL
LIN {X 0,Y 256.119,Z 323.58,A -85,B 0,C 180,E1 -18682.458,E2 -18682.458} C_VEL
LIN {X 0,Y 256.058,Z 323.563,A -85,B 0,C 180,E1 -18686.706,E2 -18686.706} C_VEL
LIN {X 0,Y 256.047,Z 323.584,A -85,B 0,C 180,E1 -18690.392,E2 -18690.392} C_VEL
LIN {X 0,Y 256.122,Z 323.575,A -85,B 0,C 180,E1 -18694.889,E2 -18694.889} C_VEL
LIN {X 0,Y 256.115,Z 323.579,A -85,B 0,C 180,E1 -18699.101,E2 -18699.101} C_VEL
LIN {X 0,Y 256.204,Z 323.571,A -85,B 0,C 180,E1 -18704.079,E2 -18704.079} C_VEL
LIN {X 0,Y 256.265,Z 323.562,A -85,B 0,C 180,E1 -18708.932,E2 -18708.932} C_VEL
LIN {X 0,Y 256.457,Z 323.524,A -85,B 0,C 180,E1 -18712.157,E2 -18712.157} C_VEL
LIN {X 0,Y 256.411,Z 323.528,A -85,B 0,C 180,E1 -18716.858,E2 -18716.858} C_VEL
LIN {X 0,Y 256.658,Z 323.508,A -85,B 0,C 180,E1 -18718.975,E2 -18718.975} C_VEL
LIN {X 0,Y 256.313,Z 323.558,A -85,B 0,C 180,E1 -18719.85,E2 -18719.85} C_VEL
LIN {X 0,Y 254.873,Z 323.735,A -85,B 0,C 180,E1 -18721.139,E2 -18721.139} C_VEL
LIN {X 0,Y 250.369,Z 324.295,A -85,B 0,C 180,E1 -18724.142,E2 -18724.142} C_VEL
LIN {X 0,Y 249.377,Z 324.42,A -85,B 0,C 180,E1 -18725.49,E2 -18725.49} C_VEL
LIN {X 0,Y 249.343,Z 324.416,A -85,B 0,C 180,E1 -18725.947,E2 -18725.947} C_VEL
LIN {X 0,Y 249.376,Z 324.414,A -85,B 0,C 180,E1 -18729.479,E2 -18729.479} C_VEL
LIN {X 0,Y 249.175,Z 324.436,A -85,B 0,C 180,E1 -18734.706,E2 -18734.706} C_VEL
LIN {X 0,Y 249.109,Z 324.436,A -85,B 0,C 180,E1 -18738.08,E2 -18738.08} C_VEL
LIN {X 0,Y 249.073,Z 324.453,A -85,B 0,C 180,E1 -18741.52,E2 -18741.52} C_VEL
LIN {X 0,Y 249.056,Z 324.461,A -85,B 0,C 180,E1 -18745.45,E2 -18745.45} C_VEL
LIN {X 0,Y 249.03,Z 324.461,A -85,B 0,C 180,E1 -18748.975,E2 -18748.975} C_VEL
LIN {X 0,Y 249.022,Z 324.458,A -85,B 0,C 180,E1 -18752.428,E2 -18752.428} C_VEL
LIN {X 0,Y 249.005,Z 324.463,A -85,B 0,C 180,E1 -18756.35,E2 -18756.35} C_VEL
LIN {X 0,Y 248.967,Z 324.475,A -85,B 0,C 180,E1 -18760.486,E2 -18760.486} C_VEL
LIN {X 0,Y 248.978,Z 324.455,A -85,B 0,C 180,E1 -18764.886,E2 -18764.886} C_VEL
LIN {X 0,Y 249.01,Z 324.488,A -85,B 0,C 180,E1 -18765.948,E2 -18765.948} C_VEL
LIN {X 0,Y 251.546,Z 333.076,A -85,B 0,C 180,E1 -18770.4,E2 -18770.4} C_VEL
LIN {X 0,Y 252.796,Z 337.439,A -85,B 0,C 180,E1 -18772.394,E2 -18772.394} C_VEL
LIN {X 0,Y 255.242,Z 341.746,A -85,B 0,C 180,E1 -18773.065,E2 -18773.065} C_VEL
LIN {X 0,Y 261.219,Z 352.861,A -85,B 0,C 180,E1 -18774.642,E2 -18774.642} C_VEL
LIN {X 0,Y 267.574,Z 365.552,A -85,B 0,C 180,E1 -18776.227,E2 -18776.227} C_VEL
LIN {X 0,Y 271.326,Z 374.206,A -85,B 0,C 180,E1 -18777.149,E2 -18777.149} C_VEL
LIN {X 0,Y 274.119,Z 390.82,A -85,B 0,C 180,E1 -18778.143,E2 -18778.143} C_VEL
LIN {X 0,Y 271.714,Z 446.905,A -85,B 0,C 180,E1 -18779.641,E2 -18779.641} C_VEL
LIN {X 0,Y 270.376,Z 460.323,A -85,B 0,C 180,E1 -18780.267,E2 -18780.267} C_VEL
LIN {X 0,Y 268.395,Z 473.04,A -85,B 0,C 180,E1 -18781.134,E2 -18781.134} C_VEL
LIN {X 0,Y 266.159,Z 484.806,A -85,B 0,C 180,E1 -18782.266,E2 -18782.266} C_VEL
LIN {X 0,Y 263.459,Z 496.157,A -85,B 0,C 180,E1 -18783.675,E2 -18783.675} C_VEL
LIN {X 0,Y 260.881,Z 506.396,A -85,B 0,C 180,E1 -18785.321,E2 -18785.321} C_VEL
LIN {X 0,Y 258.06,Z 515.639,A -85,B 0,C 180,E1 -18787.166,E2 -18787.166} C_VEL
LIN {X 0,Y 255.609,Z 523.264,A -85,B 0,C 180,E1 -18789.059,E2 -18789.059} C_VEL
LIN {X 0,Y 253.32,Z 530.747,A -85,B 0,C 180,E1 -18791.396,E2 -18791.396} C_VEL
LIN {X 0,Y 251.18,Z 536.794,A -85,B 0,C 180,E1 -18793.753,E2 -18793.753} C_VEL
LIN {X 0,Y 249.501,Z 541.606,A -85,B 0,C 180,E1 -18796.149,E2 -18796.149} C_VEL
LIN {X 0,Y 248.323,Z 545.323,A -85,B 0,C 180,E1 -18798.575,E2 -18798.575} C_VEL
LIN {X 0,Y 247.744,Z 547.255,A -85,B 0,C 180,E1 -18800.202,E2 -18800.202} C_VEL
LIN {X 0,Y 247.333,Z 548.773,A -85,B 0,C 180,E1 -18801.834,E2 -18801.834} C_VEL
LIN {X 0,Y 246.883,Z 550.543,A -85,B 0,C 180,E1 -18805.102,E2 -18805.102} C_VEL
LIN {X 0,Y 246.922,Z 550.786,A -85,B 0,C 180,E1 -18808.37,E2 -18808.37} C_VEL
LIN {X 0,Y 246.984,Z 550.283,A -85,B 0,C 180,E1 -18810.001,E2 -18810.001} C_VEL
LIN {X 0,Y 246.959,Z 549.375,A -85,B 0,C 180,E1 -18811.632,E2 -18811.632} C_VEL
LIN {X 0,Y 246.903,Z 548.064,A -85,B 0,C 180,E1 -18813.265,E2 -18813.265} C_VEL
LIN {X 0,Y 246.953,Z 546.102,A -85,B 0,C 180,E1 -18815.083,E2 -18815.083} C_VEL
LIN {X 0,Y 247.121,Z 542.854,A -85,B 0,C 180,E1 -18817.354,E2 -18817.354} C_VEL
LIN {X 0,Y 247.552,Z 538.258,A -85,B 0,C 180,E1 -18819.809,E2 -18819.809} C_VEL
LIN {X 0,Y 248.406,Z 531.261,A -85,B 0,C 180,E1 -18822.667,E2 -18822.667} C_VEL
LIN {X 0,Y 249.677,Z 523.682,A -85,B 0,C 180,E1 -18825.094,E2 -18825.094} C_VEL
LIN {X 0,Y 251.019,Z 515.93,A -85,B 0,C 180,E1 -18827.098,E2 -18827.098} C_VEL
LIN {X 0,Y 252.37,Z 506.223,A -85,B 0,C 180,E1 -18829.14,E2 -18829.14} C_VEL
LIN {X 0,Y 254.008,Z 495.875,A -85,B 0,C 180,E1 -18830.87,E2 -18830.87} C_VEL
